(* IEC 61131-3 sources: CS_4_Aufzugsteuerung/src/Stations/CP112/Steuerung/Class/_VaranDriveBase, 1 file *)

(* ---- _VaranDriveBase.st ---- *)
#ifndef _T_VARANDRIVEBASE_H
#define _T_VARANDRIVEBASE_H

#define VAC011_DEVICE_ID		              1005					// device id of VAC011
#define VAC012_DEVICE_ID		              1061					// device id of VAC012
#define VAC013_DEVICE_ID		              1075					// device id of VAC012

#define DIASDRIVE_MAXI_DEVICE_ID          1070          // device id of Dias Drive Maxi
#define DIASDRIVE_MINI_DEVICE_ID          1071          // device id of Dias Drive Mini

//#define DIASDRIVE_WaitTime_ns		            1ms * 1000 * 1000	//time in ns to send next DO in async mode

#define DIASDRIVE_OFFSET_Axis		            16#40							// memory for every axis (offset for axis 1 is 0, for axis 2 is 16#40..)
#define DIASDRIVE_OFFSET_AxisRead	          16#20							//Offset to read data of one axis
#define DIASDRIVE_OFFSET_FAST_AXIS_WRITE    16#C0
#define DIASDRIVE_OFFSET_FAST_AXIS_READ     DIASDRIVE_OFFSET_FAST_AXIS_WRITE + 16#22

#define DIASDRIVE_QUIT_ERROR_WAIT_TIME    50  // in ms

// drive address mapping
#define DIASDRIVE_ADR_ALT_BUF             16#0000  // memory offset for alternating buffer of drive
#define DIASDRIVE_ADR_SERVICE             16#1000  // memory offset for service data of drive
#define DIASDRIVE_ADR_PLL                 16#2000  // memory offset for PLL of drive
#define DIASDRIVE_ADR_LVDS_BUS            16#3000  // memory offset for lvds bus interface of drive
#define DIASDRIVE_ADR_LVDS_DIAG           16#4000  // memory offset for lvds diagnostic of drive

#define DIASDRIVE_ADR_INPUTS              16#4900  // memory offset of digital inputs

#define DIASDRIVE_ADR_OFFSET_CHANNEL      16#0800  // memory for every channel
#define DIASDRIVE_ADR_OFFSET_AXIS         16#0200  // memory for every axis

#define DIASDRIVE_ADR_AXIS_WR_OFFSET      16#0000  // offset to access write data
#define DIASDRIVE_ADR_AXIS_RD_OFFSET      16#0100  // offset to access read data

#define DIASDRIVE_ADR_ALT_BUF_RD_OFFSET   16#0400
#define DIASDRIVE_ADR_ALT_BUF_WR_OFFSET   16#0000

#define DIASDRIVE_ADR_SERVICE_READ        16#0030
#define DIASDRIVE_ADR_SERVICE_WRITE       16#0000

#define DIASDRIVE_MAX_AXIS                8
#define DIASDRIVE_MAX_AXIS_PER_MODULE     3
#define DIASDRIVE_MAX_AXIS_300            3 // with dias drive 300 only up to 3 axis possible

#define WRITETIME_TO_DPRAM                1000 // time in ns to write data to manager dpram

#endif // _T_VARANDRIVEBASE_H

(*!
<Class
	Name               = "_VaranDriveBase"
	Revision           = "1.69"
	RealtimeTask       = "false"
	CyclicTask         = "false"
	BackgroundTask     = "false"
	Sigmatek           = "true"
	OSInterface        = "false"
	HighPriority       = "false"
	Automatic          = "false"
	UpdateMode         = "Prescan"
	IconPath           = ".\Class\Varan_16x16.ico"
	SharedCommandTable = "true"
	Objectsize         = "(584,120)"
	Comment            = "class for VAC011, VAC012 and DiasDrive Mini/Maxi varan interface card">
	<Channels>
		<Server Name="CRC_ErrorCounter" Visualized="true" Initialize="false" WriteProtected="true" Retentive="false" Comment="counts CRC error of all 3 axis"/>
		<Server Name="Input1" Visualized="false" Initialize="false" WriteProtected="true" Retentive="false" Comment="State of digital input 1 of drive&#13;&#10;&#13;&#10;-1..input information not available&#13;&#10; 0..input is low&#13;&#10; 1..input is high"/>
		<Server Name="Input2" Visualized="false" Initialize="false" WriteProtected="true" Retentive="false" Comment="State of digital input 2 of drive&#13;&#10;&#13;&#10;-1..input information not available&#13;&#10; 0..input is low&#13;&#10; 1..input is high"/>
		<Server Name="Input3" Visualized="false" Initialize="false" WriteProtected="true" Retentive="false" Comment="State of digital input 3 of drive&#13;&#10;&#13;&#10;-1..input information not available&#13;&#10; 0..input is low&#13;&#10; 1..input is high"/>
		<Server Name="Input4" Visualized="false" Initialize="false" WriteProtected="true" Retentive="false" Comment="State of digital input 4 of drive&#13;&#10;&#13;&#10;-1..input information not available&#13;&#10; 0..input is low&#13;&#10; 1..input is high"/>
		<Server Name="Input5" Visualized="false" Initialize="false" WriteProtected="true" Retentive="false" Comment="State of digital input 5 of drive&#13;&#10;&#13;&#10;-1..input information not available&#13;&#10; 0..input is low&#13;&#10; 1..input is high"/>
		<Server Name="Input6" Visualized="false" Initialize="false" WriteProtected="true" Retentive="false" Comment="State of digital input 6 of drive&#13;&#10;&#13;&#10;-1..input information not available&#13;&#10; 0..input is low&#13;&#10; 1..input is high"/>
		<Server Name="Input7" Visualized="false" Initialize="false" WriteProtected="true" Retentive="false" Comment="State of digital input 7 of drive&#13;&#10;&#13;&#10;-1..input information not available&#13;&#10; 0..input is low&#13;&#10; 1..input is high"/>
		<Server Name="Input8" Visualized="false" Initialize="false" WriteProtected="true" Retentive="false" Comment="State of digital input 8 of drive&#13;&#10;&#13;&#10;-1..input information not available&#13;&#10; 0..input is low&#13;&#10; 1..input is high"/>
		<Server
			Name           = "RetryCounter"
			Initialize     = "false"
			Visualized     = "true"
			WriteProtected = "true"
			Comment        = "retry counter of varan module">
		</Server>
		<Server
			Name           = "State"
			Initialize     = "false"
			Visualized     = "true"
			WriteProtected = "true">
		</Server>
		<Server Name="Synchron" Visualized="true" Initialize="false" WriteProtected="true" Retentive="false"/>
		<Server Name="VaranOut_1" Class="Hub_Base" Visualized="true" Initialize="false" WriteProtected="true" Retentive="false"/>
		<Client Name="FetchDigitalInputs" Required="false" Internal="false" DefValue="0" Comment="Client is set as init value.&#13;&#10;a value &lt;&gt; 0 means the digital inputs of the drive are fetched synchronously and displayed on the Servers Input1 to Input8"/>
		<Client Name="Hub_Base0" Required="true" Internal="true"/>
		<Client Name="VaranTimeMultiplier" Required="false" Internal="false" Comment="multiplier of varan time as init value."/>
	</Channels>
	<RevDoku>
		<Owner Company="Sigmatek" Author="RamAnd"/>
		<Dokumentation Revision="1.69" Date="16.10.2023" Author="LanSte" Company="Sigmatek" Description="Added GetRequiredWaitTime. If this method is overwritten, the class will wait for for an required module in the init()"/>
		<Dokumentation Revision="1.68" Date="15.06.2022" Author="RamAnd" Company="Sigmatek" Description="Added new Server HardwareVersion to show the hardware version of the VARAN type label."/>
		<Dokumentation Revision="1.67" Date="07.04.2020" Author="EisMic" Company="Sigmatek" Description="Changed comment of client &quot;UserAction&quot; in Varan_Base class."/>
		<Dokumentation Revision="1.66" Date="09.12.2019" Author="LanSte" Company="Sigmatek" Description="Added Server ProtocolVersion. InterframeGap is included in the resource calculation."/>
		<Dokumentation Revision="1.65" Date="30.01.2018" Author="RamAnd" Company="Sigmatek" Description="Class is using constant VM_MULTIVARAN_ADD_DO_INTO_DOL now from VaranManager_Base.h file instead of own define section."/>
		<Dokumentation Revision="1.64" Date="06.02.2017" Author="PieSte" Company="Sigmatek" Description="Changed &quot;Online&quot; server behavior to set online first if cyclic data is valid due to SA35740.&#13;&#10;Corrected an error that MDD100 drives are not initialized if Payload is active."/>
		<Dokumentation Revision="1.63" Date="02.09.2016" Author="ZoePat" Company="Sigmatek" Description="Corrected error with asyncron communication, that could overwrite realtime data for 1 cycle if a SDD3xx was used with VarantimeMultiplier &gt; 1."/>
		<Dokumentation Revision="1.62" Date="10.05.2016" Author="RamAnd" Company="Sigmatek" Description="Suppressed warning that would occur with target ARM on compiler version 30 or higher."/>
		<Dokumentation Revision="1.61" Date="02.05.2016" Author="EisMic" Company="Sigmatek" Description="Corrected an error that SDD115 and SDD120 were not initialized."/>
		<Dokumentation Revision="1.60" Date="04.04.2016" Author="EisMic" Company="Sigmatek" Description="Corrected error in initialisation which leads to an error that the drive is not initialized."/>
		<Dokumentation Revision="1.59" Date="17.02.2016" Author="EisMic" Company="Sigmatek" Description="Prescalersettings were not set correctly when Payload is active."/>
		<Dokumentation Revision="1.58" Date="24.08.2015" Author="EisMic" Company="Sigmatek" Description="DataObjects are now installed in UpdateCy and are added to DOList in UpdateRt if the OS supports the new interface method. Version 16#1003 or higher of the pMultiVaran-Interface is needed to use this feature."/>
		<Dokumentation Revision="1.57" Date="17.06.2015" Author="PieSte" Company="Sigmatek" Description="Corrected function Varan_HwDisconnect() to set dataobjects off."/>
		<Dokumentation Revision="1.56" Date="24.03.2015" Author="EisMic" Company="Sigmatek" Description="Check pointer p_NodeInfo for validity in method GetRetryTimeout due to access exception error if method Varan_HWDisconnect is called and no hardware was available."/>
		<Dokumentation Revision="1.55" Date="30.07.2014" Author="RamAnd" Company="Sigmatek" Description="Loop to check for retries could have caused a crash, if the drive wasn&apos;t initialized so far."/>
		<Dokumentation Revision="1.54" Date="07.07.2014" Author="LanSte" Company="Sigmatek" Description="Added support for reading hardware diagnosis via newinst cmd: CMD_GET_HARDWARE_DIAGNOSE "/>
		<Dokumentation Revision="1.53" Date="04.07.2014" Author="PieSte" Company="Sigmatek" Description="Saved client FetchDigitalInputs to TempFetchDigitalInputs to avoid an access exception if it was changed during run."/>
		<Dokumentation Revision="1.52" Date="07.05.2014" Author="LanSte" Company="Sigmatek" Description="Minimized the interface request via CILGET by useing private pointers to reduce time in init."/>
		<Dokumentation Revision="1.51" Date="06.03.2014" Author="RamAnd" Company="Sigmatek" Description="Changed offset of SyncOut 1 (62,5µs) to be synchron with the SyncOut 0 to prevent inconsistent data in the drive firmware."/>
		<Dokumentation Revision="1.50" Date="12.02.2014" Author="ZoePat" Company="Sigmatek" Description="ExtendedAxis for Axis2 of SDD210 and SDD215 din&apos;t work."/>
		<Dokumentation Revision="1.40" Date="20.01.2014" Author="RamAnd&#13;&#10;PieSte" Company="Sigmatek" Description="Success of GetSyncParameter and SetSyncParameter couldn&apos;t be ensured because the return value wasn&apos;t initialized if the method succeeds.&#13;&#10;Add TaskDelay 15ms in Varan_HwConnect to initialize the Hardware."/>
		<Dokumentation Revision="1.30" Date="05.12.2013" Author="Peeale" Company="Sigmatek" Description="Added payload support; ISO-DOs now start in RT-task to work also on ARM-CPUs;"/>
		<Dokumentation Revision="1.23" Date="18.07.2012" Author="ObeChr" Company="Sigmatek" Description="Implemented time measurement for internal tests in methods UpdateRt, UpdateRtPostScan and UpdateCy"/>
		<Dokumentation Revision="1.22" Date="25.01.2012" Author="ZoePat" Company="Sigmatek" Description="Corrected usage of ENUM types."/>
		<Dokumentation Revision="1.21" Date="09.11.2011" Author="RamAnd" Company="Sigmatek" Description="The memory initialisation of last change has been done too late (after new data was already set)."/>
		<Dokumentation Revision="1.20" Date="16.08.2011" Author="PibPet" Company="Sigmatek" Description="Fixed Problem with the Initialisation from the Drive. Reinit the Memory before sending."/>
		<Dokumentation Revision="1.19" Date="05.07.2011" Author="RamAnd" Company="Sigmatek" Description="Fixed problems in intialisation of SDD drives with less than 3 axis."/>
		<Dokumentation Revision="1.18" Date="14.06.2011" Author="RamAnd" Company="Sigmatek" Description="Fixed crash, when a MDD100 is exchanged with a SDD300 or the other way round."/>
		<Dokumentation Revision="1.17" Date="31.05.2011" Author="RamAnd" Company="Sigmatek" Description="Added possibility to read out the digital inputs of the drive synchronously."/>
		<Dokumentation Revision="1.16" Date="31.05.2011" Author="RamAnd" Company="Sigmatek" Description="DataObjects for VARAN communication are now created and started in the corresponding tasks (ISO-DOs in RT and ASY-DOs in CY) instead of creating and starting all DOs in the connect-callback."/>
		<Dokumentation Revision="1.15" Date="18.05.2011" Author="RamAnd" Company="Sigmatek" Description="After the Online-Server changed to 1, it was possible that the synchron values (like actual position) took 1 more realtime cycle to be shown by the class."/>
		<Dokumentation Revision="1.14" Date="04.01.2011" Author="BleErn" Company="Sigmatek" Description="Added Client Transparent that allows to disable a VARAN-HW-Class"/>
		<Dokumentation Revision="1.13" Date="14.02.2011" Author="BleErn" Company="Sigmatek" Description="Fixed problems with asynchronous communication"/>
		<Dokumentation Revision="1.12" Date="07.12.2010" Author="RamAnd" Company="Sigmatek" Description="Fixed problems in initialisation, when device is plugged in and out within a short time."/>
		<Dokumentation Revision="1.11" Date="25.10.2010" Author="BleErn" Company="Sigmatek" Description="Safety input of VAC013 did not trigger correct errors because of a incorrect comparison of HW-ID"/>
		<Dokumentation Revision="1.10" Date="13.08.2010" Author="BleErn" Company="Sigmatek" Description="Removed an irritating comment from implementation"/>
		<Dokumentation Revision="1.9" Date="10.08.2010" Author="Ramand" Company="Sigmatek" Description="Added support for SDD115"/>
		<Dokumentation Revision="1.8" Date="02.06.2010" Author="BleErn / RamAnd" Company="Sigmatek" Description="Optimization of UpdateRtPostScan method.&#13;&#10;Added support for SDD210"/>
		<Dokumentation Revision="1.7" Date="10.03.2010" Author="RamAnd" Company="Sigmatek" Description="Added serial number validation"/>
		<Dokumentation Revision="1.6" Date="17.05.2010" Author="RamAnd" Company="Sigmatek" Description="Changed defines to avoid compiler warning &quot;Identical Redefinition&quot;"/>
		<Dokumentation Revision="1.5" Date="26.02.2010" Author="RamAnd" Company="Sigmatek" Description="Added support for VAC013"/>
		<Dokumentation Revision="1.4" Date="15.02.2010" Author="RamAnd" Company="Sigmatek" Description="Class works now also with SDD215"/>
		<Dokumentation Revision="1.3" Date="15.01.2010" Author="RamAnd" Company="Sigmatek" Description="Removed Client AxisAvailable. The available axis are now automatically detected."/>
		<Dokumentation Revision="1.2" Date="03.12.2009" Author="RamAnd" Company="Sigmatek" Description="Improved comment on client &quot;AxisAvailable&quot;."/>
		<Dokumentation Revision="1.1" Date="09.11.2009" Author="RamAnd" Company="Sigmatek" Description="Login of VaranRtPostScan did not work properly if the init of the _VaranDriveBase has been called before the VaranManager-Init."/>
		<Dokumentation Revision="1.0" Date="06.10.2009" Author="RamAnd" Company="Sigmatek" Description="Error in Init has been solved (could have led to a VARAN FATAL ERROR)"/>
	</RevDoku>
	<Network Name="_VaranDriveBase">
		<!-- List of Components in this network -->
		<Components>
			<Object
				Name       = "_base"
				Class      = "Varan_Base"
				Position   = "(240,120)"
				Visualized = "true">
				<Channels>
					<Server Name="ConnectCounter"/>
					<Server Name="DeviceAddress"/>
					<Server Name="DeviceID"/>
					<Server Name="DiagControl"/>
					<Server Name="FaultCounter"/>
					<Server Name="HardwareVersion"/>
					<Server Name="Online"/>
					<Server Name="ProtocolVersion"/>
					<Server Name="Release"/>
					<Server Name="RetryCounter"/>
					<Server Name="RXLost"/>
					<Server Name="SerialNo"/>
					<Server Name="State"/>
					<Server Name="TXLost"/>
					<Server Name="ValidateSerNo"/>
					<Server Name="VendorID"/>
					<Client Name="Required" Value="1"/>
					<Client Name="SerNoValidation"/>
					<Client Name="TimeBase" Value="0"/>
					<Client Name="TimeBaseOffset" Value="0"/>
					<Client Name="To_MultiTask"/>
					<Client Name="To_StdLib"/>
					<Client Name="Transparent"/>
					<Client Name="UserAction"/>
					<Client Name="VaranIn"/>
				</Channels>
			</Object>
			<Object
				Name       = "Hub_Base0"
				Class      = "Hub_Base"
				Position   = "(870,780)"
				Visualized = "true">
				<Channels>
					<Server Name="Control"/>
					<Client Name="Splitter_Place" Value="0"/>
					<Client Name="VaranIn"/>
				</Channels>
			</Object>
		</Components>
		<Comments>
		</Comments>
		<!-- List of Connections in this network -->
		<Connections>
			<Connection Source="this.State" Destination="_base.State" Vertices="(1468,210),(724,210),"/>
			<Connection Source="this.Online" Destination="_base.Online" Vertices="(1468,270),(724,270),"/>
			<Connection Source="this.Release" Destination="_base.Release" Vertices="(1468,330),(724,330),"/>
			<Connection Source="this.DeviceAddress" Destination="_base.DeviceAddress" Vertices="(1468,450),(724,450),"/>
			<Connection Source="_base.VaranIn" Destination="this.VaranIn" Vertices="(240,210),(38,210),"/>
			<Connection Source="_base.Required" Destination="this.Required" Vertices="(240,270),(38,270),"/>
			<Connection Source="this.VendorID" Destination="_base.VendorID" Vertices="(1468,510),(724,510),"/>
			<Connection Source="this.DeviceID" Destination="_base.DeviceID" Vertices="(1468,570),(724,570),"/>
			<Connection Source="_base.UserAction" Destination="this.UserAction" Vertices="(240,330),(38,330),"/>
			<Connection Source="Hub_Base0.VaranIn" Destination="_base.State" Vertices="(870,870),(810,870),(810,210),(724,210),"/>
			<Connection Source="this.VaranOut_1" Destination="Hub_Base0.Control" Vertices="(1468,1470),(1296,870),"/>
			<Connection Source="this.RetryCounter" Destination="_base.RetryCounter" Vertices="(1468,690),(724,690),"/>
			<Connection Source="this.Hub_Base0" Destination="Hub_Base0.Control"/>
			<Connection Source="this.SerialNo" Destination="_base.SerialNo" Vertices="(1468,630),(724,630),"/>
			<Connection Source="_base.SerNoValidation" Destination="this.SerNoValidation" Vertices="(240,390),(38,390),"/>
			<Connection Source="this.ValidateSerNo" Destination="_base.ValidateSerNo" Vertices="(1468,750),(724,750),"/>
			<Connection Source="_base.Transparent" Destination="this.Transparent" Vertices="(240,450),(38,450),"/>
			<Connection Source="this.ProtocolVersion" Destination="_base.ProtocolVersion" Vertices="(1468,810),(724,1110),"/>
			<Connection Source="this.HardwareVersion" Destination="_base.HardwareVersion" Vertices="(1468,390),(724,390),"/>
		</Connections>
		<!-- Headerfiles -->
		<Options>
		</Options>
	</Network>
</Class>
*)
#pragma using Varan_Base

_VaranDriveBase : CLASS
: Varan_Base
	TYPE
	  t_AxisState :
	  (
	    _NotUsed,
	    _NoInit,
	    _InitOk,
	    _NoParaList,
	    _NotSynchron,
	    _AxisOk
	  )$USINT;
	  t_ParaState :
	  (
	    _SendExecution,
	    _ResetExecution,
	    _Wait4Response,
	    _IdleState,
	    _GotValueForExecution
	  )$UDINT;
#pragma pack(push, 1)
	  t_ParaList : STRUCT
	    us_number : USINT;
	    sd_value : DINT;
	  END_STRUCT;
#pragma pack(pop)
#pragma pack(push, 1)
	  t_ReadValuePtr : STRUCT  //! <Type Public="true" Name="t_ReadValuePtr"/>
	    a_SyncValues : ARRAY [0..4] OF DINT;
	    bs_InputStates : BSINT
	    [
	      1 OptionBoardInputState,
	    ];
	  END_STRUCT;
#pragma pack(pop)
#pragma pack(push, 1)
	  t_WriteValuePtr : STRUCT  //! <Type Public="true" Name="t_WriteValuePtr"/>
	    a_SyncValues : ARRAY [0..4] OF DINT;
	  END_STRUCT;
#pragma pack(pop)
	  t_AxisData : STRUCT
	    e_AxisState : t_AxisState;
	    us_ParaReady : t_ParaState;
	    sd_Asyncdata : DINT;
	    sd_ObjectError : DINT;
	    b_ListActive : BOOL;
	    p_ParaList : ^t_ParaList;
	    ui_ParaListCnt : UINT;
	    ud_CRCError : UDINT;
	    ud_DOLength : UDINT;
	    b_ExtendedAxis : DINT;
	    b_FastAxis : DINT;
	    b_OldToggleState : DINT;
	    s_ReadValues : t_ReadValuePtr;
	    s_WriteValues : t_WriteValuePtr;
	  END_STRUCT;
#pragma pack(push, 1)
	  t_DataReadOneAxis : STRUCT
	    us_ReceiveState : BSINT
	    [
	      1 ExecutedObjectTransfer,
	      2 CRC_Error,
	      4 OnlineToolWriteOk,
	    ];
	    us_Reserved1 : USINT;
	    us_DigitalIO : USINT;
	    us_TransmitControl : BSINT
	    [
	      1 ToggleBit,
	      2 ErrorInObjectHandling,
	      3 Warning,
	      4 ErrorBit,
	      5 SyncLocked,
	      6 MainsApplied,
	      7 ExternalLock,
	      8 notused,
	    ];
	    sd_ObjectValue : DINT;
	    sd_Value6 : DINT;
	    sd_Value7 : DINT;
	    sd_Value8 : DINT;
	    sd_Value9 : DINT;
	    sd_Value10 : DINT;
	  END_STRUCT;
#pragma pack(pop)
#pragma pack(push, 1)
	  t_DataWriteAsync : STRUCT
	    us_TransmitExecution : BSINT
	    [
	      1 StartObjectTransfer,
	      2 RepeatObjectTransfer,
	      3 EnableValue3_5,
	      4 ClearOnlineToolWriteOk,
	    ];
	    us_Reserved1 : USINT;
	    us_DriveControl : BSINT
	    [
	      1 ToggleBit,
	      2 ReadWriteObject,
	      3 InitCommunicatian,
	      4 EnableInput1,
	      5 UnlockInput1,
	      6 UnlockBrake,
	      7 InterfaceComError,
	      8 NoSetPoint,
	    ];
	    us_ObjectAddress : USINT;
	    sd_ObjectValue : DINT;
	  END_STRUCT;
#pragma pack(pop)
#pragma pack(push, 1)
	  t_DataWriteOneAxis : STRUCT
	    us_TransmitExecution : BSINT
	    [
	      1 StartObjectTransfer,
	      2 RepeatObjectTransfer,
	      3 EnableValue3_5,
	      4 ClearOnlineToolWriteOk,
	    ];
	    us_Reserved1 : USINT;
	    us_DriveControl : BSINT
	    [
	      1 ToggleBit,
	      2 ReadWriteObject,
	      3 InitCommunication,
	      4 EnableInput1,
	      5 UnlockInput1,
	      6 UnlockBrake,
	      7 InterfaceComError,
	      8 NoSetPoint,
	    ];
	    us_ObjectAddress : USINT;
	    sd_ObjectValue : DINT;
	    sd_Value1 : DINT;
	    sd_Value2 : DINT;
	    sd_Value3 : DINT;
	    sd_Value4 : DINT;
	    sd_Value5 : DINT;
	  END_STRUCT;
#pragma pack(pop)
#pragma pack(push, 1)
	  t_FastAxisRead : STRUCT
	    us_DigInOut : USINT;
	    us_TrasmittControl : USINT;
	    sd_Value8 : DINT;
	    sd_Value9 : DINT;
	    sd_Value10 : DINT;
	  END_STRUCT;
#pragma pack(pop)
#pragma pack(push, 1)
	  t_FastAxisWrite : STRUCT
	    us_TransmittExecution : BSINT
	    [
	      5 EnableType2,
	      6 DirectAccess,
	    ];
	    us_Reserved1 : USINT;
	    us_DriveControl : USINT;
	    us_Reserved2 : USINT;
	    sd_Value3 : DINT;
	    sd_Value4 : DINT;
	    sd_Value5 : DINT;
	  END_STRUCT;
#pragma pack(pop)
#pragma pack(push, 1)
	  t_DOFastAxis : STRUCT
	    p_Handle : ^LSL_VARANFRAME;
	    p_DOSettings : ^t_VaranDOSettingsRdWr;
	    p_DataRead : ^t_FastAxisRead;
	    p_DataWrite : ^t_FastAxisWrite;
	    us_OldRetryCounter : USINT;
	  END_STRUCT;
#pragma pack(pop)
	  t_DOOneAxis : STRUCT
	    p_Handle : ^LSL_VARANFRAME;
	    p_DOSettings : ^t_VaranDOSettingsRdWr;
	    p_DataRead : ^t_DataReadOneAxis;
	    p_DataWrite : ^t_DataWriteOneAxis;
	    AsyDataTemp : t_DataWriteOneAxis;
	    b_NewAsyDataTemp : BOOL;
	    us_OldRetryCounter : USINT;
	  END_STRUCT;
#pragma pack(push, 1)
	  t_DrivePLLRd : STRUCT
	    SystemPeriodTime : UINT;
	    Reserved1 : UINT;
	    MaxCountValue : UINT;
	    Reserved2 : UINT;
	    DriveCycleCounter : UINT;
	    StatusRegister : BSINT
	    [
	      1 PLL_Locked,
	    ];
	    Reserved3 : SINT;
	    SyncOut1Offset : UINT;
	    Reserved4 : UINT;
	  END_STRUCT;
#pragma pack(pop)
#pragma pack(push, 1)
	  t_DrivePLLWr : STRUCT
	    SystemPeriodTime : UINT;
	    Reserved1 : UINT;
	  END_STRUCT;
#pragma pack(pop)
	  t_InitSSW :
	  (
	    _SetDataObjectOn,
	    _SetInitAxis,
	    _WaitInit,
	    _SetFinishInit,
	    _SetExecuteBack,
	    _GetFinishInit,
	    _CyIdle
	  )$UDINT;
#pragma pack(push, 1)
	  t_newASYRead : STRUCT
	    sd_ObjectValue : DINT;
	    us_TransmitControl : BSINT
	    [
	      1 ToggleBit,
	      2 ErrorInObjectHandling,
	      3 Warning,
	      4 ErrorBit,
	      5 SyncLocked,
	      6 MainsApplied,
	      7 ExternalLock,
	      8 notused,
	    ];
	    us_DigitalIO : USINT;
	  END_STRUCT;
#pragma pack(pop)
	  t_newASYReadArray : ARRAY [0..DIASDRIVE_MAX_AXIS-1] OF t_newASYRead;
#pragma pack(push, 1)
	  t_newASYWrite : STRUCT
	    sd_ObjectValue : DINT;
	    us_DriveControl : BSINT
	    [
	      1 ToggleBit,
	      2 ReadWriteObject,
	      3 InitCommunication,
	      4 EnableInput1,
	      5 UnlockInput1,
	      6 UnlockBrake,
	      7 InterfaceComError,
	      8 NoSetPoint,
	    ];
	    us_ObjectAddress : USINT;
	  END_STRUCT;
#pragma pack(pop)
	  t_newASYWriteArray : ARRAY [0..DIASDRIVE_MAX_AXIS-1] OF t_newASYWrite;
#pragma pack(push, 1)
	  t_newASYDO : STRUCT
	    p_Handle : ^LSL_VARANFRAME;
	    p_DOSettings : ^t_VaranDOSettingsRdWr;
	    p_DataRead : ^t_newASYReadArray;
	    p_DataWrite : ^t_newASYWriteArray;
	    us_OldRetryCounter : USINT;
	    AsyDataTemp : t_newASYWriteArray;
	    b_NewAsyDataTemp : ARRAY [0..DIASDRIVE_MAX_AXIS-1] OF BOOL;
	  END_STRUCT;
#pragma pack(pop)
#pragma pack(push, 1)
	  t_newDigInDO : STRUCT
	    p_Handle : ^LSL_VARANFRAME;
	    p_DOSettings : ^t_VaranDOSettingsRd;
	    p_DataRead : ^USINT;
	    us_OldRetryCounter : USINT;
	  END_STRUCT;
#pragma pack(pop)
#pragma pack(push, 1)
	  t_newReadDataOneAxis : STRUCT
	    Value6 : DINT;
	    Value7 : DINT;
	    Value8 : DINT;
	    Value9 : DINT;
	    Value10 : DINT;
	  END_STRUCT;
#pragma pack(pop)
#pragma pack(push, 1)
	  t_newWriteDataOneAxis : STRUCT
	    Value1 : DINT;
	    Value2 : DINT;
	    Value3 : DINT;
	    Value4 : DINT;
	    Value5 : DINT;
	  END_STRUCT;
#pragma pack(pop)
#pragma pack(push, 1)
	  t_newISODO : STRUCT
	    p_Handle : ^LSL_VARANFRAME;
	    p_DOSettings : ^t_VaranDOSettingsRdWr;
	    p_DataRead : ^t_newReadDataOneAxis;
	    p_DataWrite : ^t_newWriteDataOneAxis;
	    us_OldRetryCounter : USINT;
	  END_STRUCT;
#pragma pack(pop)
#pragma pack(push, 1)
	  t_ParaSkipOneAxis : STRUCT
	    us_No : USINT;
	    p_Values : ^USINT;
	  END_STRUCT;
#pragma pack(pop)
	  t_ParaSkipList : ARRAY [0..DIASDRIVE_MAX_AXIS-1] OF t_ParaSkipOneAxis;
	  t_RtSSW :
	  (
	    CompInitAxis,
	    CompGetSendParaList,
	    CompWaitForSynchrony,
	    CompOperational,
	    InitAxis,
	    GetSendParaList,
	    WaitForSynchrony,
	    Operational
	  )$UDINT;
	END_TYPE
  //Servers:
	CRC_ErrorCounter 	: SvrCh_DINT;
	Synchron 	: SvrCh_DINT;
	Input1 	: SvrCh_DINT;
	Input2 	: SvrCh_DINT;
	Input3 	: SvrCh_DINT;
	Input4 	: SvrCh_DINT;
	Input5 	: SvrCh_DINT;
	Input6 	: SvrCh_DINT;
	Input7 	: SvrCh_DINT;
	Input8 	: SvrCh_DINT;
	VaranOut_1 	: SvrChCmd_DINT;
  //Clients:
	Hub_Base0 	: CltChCmd_Hub_Base;
	VaranTimeMultiplier 	: CltCh_UDINT;
	FetchDigitalInputs 	: CltCh_DINT;
  //Variables:
		aAxisData : ARRAY [0..DIASDRIVE_MAX_AXIS-1] OF t_AxisData;

		aDataObjects : ARRAY [0..DIASDRIVE_MAX_AXIS-1] OF t_DOOneAxis;

		newIsoDOs : ARRAY [0..DIASDRIVE_MAX_AXIS-1] OF t_newISODO;

		newAsyDO 	: t_newASYDO;
		newDigInDO 	: t_newDigInDO;
		us_Firstscan 	: USINT;
		us_AxisNumber 	: USINT;
		e_InitSSW 	: t_InitSSW;
		b_InitOk 	: BOOL;
		ud_TimemarkInit 	: UDINT;
		ud_TimeCounter 	: UDINT;
		b_SyncEnabled 	: BOOL;
		sd_SyncOffset 	: DINT;
		ud_VaranTime 	: UDINT;
		ud_IsoStartPoint 	: UDINT;
		b_FastDODeactivate 	: BOOL;
		s_DataFastAxis 	: t_DOFastAxis;
		RwFastSpeed 	: t_FastAxisWrite;
		s_SkipParameter 	: t_ParaSkipList;
		AxisAvailableHW : BDINT
		[
		];

		ExtendedAxisSettings : BDINT
		[
		];

		FastAxisSettings : BDINT
		[
		];

		b_CompatibilityMode 	: BOOL;			//! <Variable Comment="TRUE....SDD300 series model&#13;&#10;FALSE...SDD100/5000 series model" Name="b_CompatibilityMode"/>
		pCallBackServer 	: ^UDINT;
		AxisAvailableNo 	: USINT;
		CompAxisAvailableNo 	: SINT;
		AxisAvailable100 	: USINT;
		GetCompAxisSSW 	: UDINT;
		e_RtSSW 	: t_RtSSW;
		CreatedCompDOs 	: BOOL;
		CreatedNewIsoDOs 	: BOOL;
		CreatedNewAsyDOs 	: BOOL;
		b_UpdateThisTime 	: BOOL;
		b_IsSDD21x 	: BOOL;
		b_AlreadyConnected 	: BOOL;
		DataInitFinished 	: BOOL;
		TempFetchDigitalInputs 	: BOOL;
		p_DriveMngBase 	: ^void;
		bAddDOsToListSupport 	: BOOL;			//! <Variable Comment="Flag is True if the os version supports to add DOs to DOL with multivaraninterface (MULTI_VARAN_IINSERTDOINTODOL)" Name="bAddDOsToListSupport"/>
  //Functions:
				//! <Function Comment="=================================================================================================&#13;&#10;Init for Varan Client&#13;&#10;=================================================================================================&#13;&#10;" Name="Init"/>
	FUNCTION VIRTUAL GLOBAL Init;
				//! <Function Comment="Cy - Funktion of Varan class ( called bei VaranMaster )" Name="UpdateCy"/>
	FUNCTION VIRTUAL GLOBAL UpdateCy;
				//! <Function Comment="=================================================================================================&#13;&#10;Rt - Funktion of Varan class ( called bei VaranMaster )&#13;&#10;=================================================================================================&#13;&#10;" Name="UpdateRt"/>
	FUNCTION VIRTUAL GLOBAL UpdateRt;

	FUNCTION VIRTUAL GLOBAL UpdateRtPostScan;
				//! <Function Comment="=================================================================================================&#13;&#10;Function is called if a varan module is connected&#13;&#10;=================================================================================================&#13;&#10;" Name="Varan_HwConnect"/>
	FUNCTION VIRTUAL GLOBAL Varan_HwConnect
		VAR_INPUT
			ud_data 	: UDINT;			//! <Variable Comment="data of call back" Name="Varan_HwConnect.ud_data"/>
		END_VAR
		VAR_OUTPUT
			sd_retval 	: DINT;			//! <Variable Comment="0=Ok, -1=class not okay, -2=wrong axle, -3=axle not in use, -4=varan error in data object" Name="Varan_HwConnect.sd_retval"/>
		END_VAR;
				//! <Function Comment="=================================================================================================&#13;&#10;Function is called if a varan interrupt occures&#13;&#10;=================================================================================================&#13;&#10;" Name="Varan_HwInterrupt"/>
	FUNCTION VIRTUAL GLOBAL Varan_HwInterrupt
		VAR_INPUT
			ud_reason 	: UDINT;			//! <Variable Comment="reason of interrupt" Name="Varan_HwInterrupt.ud_reason"/>
			ud_data 	: ^t_CallBackInterrupt;
		END_VAR
		VAR_OUTPUT
			sd_retval 	: DINT;
		END_VAR;
				//! <Function Comment="=================================================================================================&#13;&#10;Function is called if a varan module is disconnected&#13;&#10;=================================================================================================&#13;&#10;" Name="Varan_HwDisconnect"/>
	FUNCTION VIRTUAL GLOBAL Varan_HwDisconnect
		VAR_INPUT
			ud_data 	: UDINT;
		END_VAR
		VAR_OUTPUT
			sd_retval 	: DINT;
		END_VAR;
				//! <Function Comment="=================================================================================================&#13;&#10;Function to set all Data Objects off&#13;&#10;=================================================================================================&#13;&#10;" Name="SetDOsOff"/>
	FUNCTION VIRTUAL GLOBAL SetDOsOff;
				//! <Function Comment="=================================================================================================&#13;&#10;Function to update module retry counter&#13;&#10;=================================================================================================&#13;&#10;" Name="UpdateRetryCounter"/>
	FUNCTION VIRTUAL GLOBAL UpdateRetryCounter;
				//! <Function Comment="Check if DeviceID is supported by class" Name="CheckDeviceID"/>
	FUNCTION VIRTUAL GLOBAL CheckDeviceID
		VAR_INPUT
			ID2Check 	: UDINT;			//! <Variable Comment="VARAN DeviceID, which should be checked" Name="CheckDeviceID.ID2Check"/>
		END_VAR
		VAR_OUTPUT
			IsOK 	: BOOL;			//! <Variable Comment="TRUE...DeviceID is ok with this class&#13;&#10;FALSE..DeviceID is not ok with this class" Name="CheckDeviceID.IsOK"/>
		END_VAR;
				//! <Function Comment="[#ENGLISH]&#13;&#10;=================================================================================================&#13;&#10;Function to initailize each axle&#13;&#10;=================================================================================================&#13;&#10;[members] s_Axle[x]Data  :R/W :structure for data of one axle&#13;&#10;   s_DataObjectA[x] :R/W :structure for data object of one axle&#13;&#10;   e_InitSSW   :R/W :init ssw&#13;&#10;   ud_TimemarkInit  :W/R :timeout for init&#13;&#10;[locals] p_axle    :W/R :pointer to right axle data&#13;&#10;   p_data_object  :W/R :pointer to right axle data object information&#13;&#10;" Name="InitAxis"/>
	FUNCTION InitAxis
		VAR_INPUT
			us_AxisNo 	: USINT;			//! <Variable Comment="number of axle" Name="InitAxis.us_AxisNo"/>
		END_VAR
		VAR_OUTPUT
			sd_retval 	: DINT;
		END_VAR;
				//! <Function Comment="=================================================================================================&#13;&#10;Function to get object value state&#13;&#10;=================================================================================================&#13;&#10;" Name="GetParameterState"/>
	FUNCTION GLOBAL GetParameterState
		VAR_INPUT
			us_Axis 	: USINT;
		END_VAR
		VAR_OUTPUT
			sd_para_state 	: DINT;			//! <Variable Comment="&gt;0=Object Error, 0=ok, -1=function not ready, -2=wrong axle, -3=Axle not in use, -4=varan error in data object" Name="GetParameterState.sd_para_state"/>
		END_VAR;
				//! <Function Comment="=================================================================================================&#13;&#10;Function to set a object value&#13;&#10;=================================================================================================&#13;&#10;" Name="SetParameter"/>
	FUNCTION GLOBAL SetParameter
		VAR_INPUT
			us_Axis 	: USINT;
			us_para_nr 	: USINT;			//! <Variable Comment="number of parameter" Name="SetParameter.us_para_nr"/>
			us_rdwr 	: USINT;			//! <Variable Comment="0=read, 1=write" Name="SetParameter.us_rdwr"/>
			sd_para_value 	: DINT;			//! <Variable Comment="value of parameter (only for write)" Name="SetParameter.sd_para_value"/>
		END_VAR
		VAR_OUTPUT
			sd_retval 	: DINT;
		END_VAR;
				//! <Function Comment="=================================================================================================&#13;&#10;Function to get object value of parameter&#13;&#10;=================================================================================================&#13;&#10;" Name="GetParameter"/>
	FUNCTION GLOBAL GetParameter
		VAR_INPUT
			us_Axis 	: USINT;
		END_VAR
		VAR_OUTPUT
			sd_para_data 	: DINT;			//! <Variable Comment="value of readed parameter" Name="GetParameter.sd_para_data"/>
		END_VAR;
				//! <Function Comment="=================================================================================================&#13;&#10;Function to set parameter parameter list&#13;&#10;=================================================================================================&#13;&#10;" Name="SetParaList"/>
	FUNCTION GLOBAL SetParaList
		VAR_INPUT
			us_Axis 	: USINT;
			p_list 	: ^void;			//! <Variable Comment="pointer to parameter list" Name="SetParaList.p_list"/>
			ui_counter 	: UINT;			//! <Variable Comment="number of parameters" Name="SetParaList.ui_counter"/>
		END_VAR
		VAR_OUTPUT
			sd_retval 	: DINT;
		END_VAR;
				//! <Function Comment="=================================================================================================&#13;&#10;Function to get a synchron parameter&#13;&#10;=================================================================================================&#13;&#10;" Name="GetSyncParameter"/>
	FUNCTION GLOBAL GetSyncParameter
		VAR_INPUT
			us_Axis 	: USINT;
			us_value 	: USINT;			//! <Variable Comment="0=Value1, 1=Value2, 2=Value3, 3=Value4, 4=Value5" Name="GetSyncParameter.us_value"/>
			p_data 	: ^DINT;			//! <Variable Comment="to this pointer value is written" Name="GetSyncParameter.p_data"/>
		END_VAR
		VAR_OUTPUT
			sd_retval 	: DINT;
		END_VAR;
				//! <Function Comment="=================================================================================================&#13;&#10;Function to set a synchron Parameter&#13;&#10;=================================================================================================&#13;&#10;" Name="SetSyncParameter"/>
	FUNCTION GLOBAL SetSyncParameter
		VAR_INPUT
			us_Axis 	: USINT;
			us_value 	: USINT;
			sd_data 	: DINT;			//! <Variable Comment="data of value" Name="SetSyncParameter.sd_data"/>
		END_VAR
		VAR_OUTPUT
			sd_retval 	: DINT;
		END_VAR;

	FUNCTION InitAxisNew
		VAR_INPUT
			us_AxisNo 	: USINT;
		END_VAR
		VAR_OUTPUT
			sd_retval 	: DINT;
		END_VAR;
				//! <Function Comment="[#ENGLISH]&#13;&#10;=================================================================================================&#13;&#10;Function for parameter handling in synchron mode&#13;&#10;=================================================================================================&#13;&#10;[members] s_Axle[x]Data  :R/W :structure for data of one axle&#13;&#10;   s_DataObjectA[x] :R/W :structure for data object of one axle&#13;&#10;[locals] p_axle   :W/R :pointer to right axle data&#13;&#10;   p_DataObject :W/R :pointer to right data object for axle&#13;&#10;" Name="GetObjectValue"/>
	FUNCTION GetObjectValue
		VAR_INPUT
			us_Axis 	: USINT;
		END_VAR;

	FUNCTION GetObjectValueNew
		VAR_INPUT
			us_Axis 	: USINT;
		END_VAR;
				//! <Function Comment="=================================================================================================&#13;&#10;Function inits drive for all axes used&#13;&#10;=================================================================================================&#13;&#10;" Name="InitDrive"/>
	FUNCTION GLOBAL InitDrive;

	FUNCTION GLOBAL SetAxisOn
		VAR_INPUT
			ud_Axis 	: BDINT;
		END_VAR;
				//! <Function Comment="Function to skip parameters in the parameter list.&#13;&#10;Parameters to be skipped have to be defined via Newinst command 1" Name="SkipEntries"/>
	FUNCTION SkipEntries
		VAR_INPUT
			us_Axis 	: USINT;
			p_Axis 	: ^t_AxisData;
		END_VAR;
				//! <Function Comment="tell the drive class, the software setting and install callback (calls write-method of given server) to get available configuration" Name="StartCommunication"/>
	FUNCTION GLOBAL StartCommunication
		VAR_INPUT
			AxisExtend 	: BDINT;
			AxisFast 	: BDINT;
			pServer4CallBack 	: ^BDINT;			//! <Variable Comment="pass address of server (e.g. #MyServer) to get a callback (write-method) of this server, if the hardware is available on varan (available axis are passed as input parameter)" Name="StartCommunication.pServer4CallBack"/>
		END_VAR;

	FUNCTION GLOBAL GetAxisRdPtr
		VAR_INPUT
			AxisNr 	: DINT;			//! <Variable Comment="number of axis for which you want the pointer (1..8)" Name="GetAxisRdPtr.AxisNr"/>
		END_VAR
		VAR_OUTPUT
			pReadPara 	: ^t_ReadValuePtr;
		END_VAR;

	FUNCTION GLOBAL GetAxisWrPtr
		VAR_INPUT
			AxisNr 	: DINT;
		END_VAR
		VAR_OUTPUT
			pWritePara 	: ^t_WriteValuePtr;
		END_VAR;

	FUNCTION GLOBAL GetDriveIntState
		VAR_OUTPUT
			retcode 	: DINT;			//! <Variable Comment="0..Initialisation of Axles&#13;&#10;1..Download of Drive Parameters&#13;&#10;2..Wait until Drive is synchron with Varan&#13;&#10;3..Operational mode" Name="GetDriveIntState.retcode"/>
		END_VAR;

	FUNCTION GLOBAL ExternInitFinished;

	FUNCTION GetDriveType
		VAR_INPUT
			HWCode 	: DINT;
		END_VAR
		VAR_OUTPUT
			AxisNo 	: SINT;
		END_VAR;

	FUNCTION InstallDefaultDO;

	FUNCTION AddIsoDOsCompMode;

	FUNCTION AddIsoDOsNew;

	FUNCTION GLOBAL GetSeries
		VAR_OUTPUT
			retcode 	: USINT;
		END_VAR;

	FUNCTION GLOBAL IsSDD21x
		VAR_OUTPUT
			retcode 	: BOOL;
		END_VAR;
				//! <Function Comment="Save the passed DriveMngBase this pointer. Needed for Hardwarediagnosis." Name="SetObjectCallBack"/>
	FUNCTION GLOBAL SetObjectCallBack
		VAR_INPUT
			p_DriveMngBaseNew 	: ^void;
		END_VAR;

	FUNCTION VIRTUAL GLOBAL State::NewInst
		VAR_INPUT
			pPara 	: ^CmdStruct;
			pResult 	: ^results;
		END_VAR
		VAR_OUTPUT
			ret_code 	: iprStates;
		END_VAR;
  //Tables:
	FUNCTION @STD
		VAR_OUTPUT
			ret_code	: CONFSTATES;
		END_VAR;
	FUNCTION GLOBAL TAB @CT_;
END_CLASS;

#pragma using Hub_Base

FUNCTION VIRTUAL GLOBAL _VaranDriveBase::Init
  VAR
    sd_retval   : DINT;
  END_VAR

#ifdef IsTransparent_IS_AVAILABLE
  IF IsTransparent() THEN
    return;
  END_IF;
#endif

	//in first init phase
	if ( us_Firstscan = 1 ) then

		//-----------------------------------------------------------------------------------------------
		//init the base class
		Varan_Base::Init();

		//if an error in base class occurs return
		if ( State <> _NotInitialized ) then
			return;
		end_if;

    //Reset Flag
    bAddDOsToListSupport := FALSE;

    //bAddDosToListSupport Flag:
    //Install the isochrone dataobjects in cywork and not in the realtime task, due to the high realtime load in the first rt cycles.
    //The dataobjects are only installed an not added to the DOL in the os with the mask VARAN_DOL_NOT_INSERT_DO_INTO_DOL.
    //With the new os-function MULTI_VARAN_IINSERTDOINTODOL the Dataobjects are now added to the DOL List in the Os.
    //pMultiVaran-Interfaceversion must be equal or higher than 16#1003

    //Check interface version
    if b_PayloadSupport then
      if pMultiVaran then
        if pMultiVaran^.udVersion >= VM_MULTIVARAN_ADD_DO_INTO_DOL then
        // We have the new interface, set flag to remember it later
          bAddDOsToListSupport := TRUE;
        end_if;
      end_if;
    end_if;

    //read cycle time
    VaranTimeMultiplier := VaranTimeMultiplier.read();

    if b_PayloadSupport then
      // Payload DOs automatically use the client Timebase to set the Prescaler of the DOs
      TimeBase := VaranTimeMultiplier;
    end_if;

    if ( VaranTimeMultiplier = 0 ) then
      VaranTimeMultiplier := 1;
    end_if;

    //because on startup we need no waittime for bootloader
    us_AxisNumber := 1;

    //get varan time and calculate offset for sync
    ud_VaranTime := VaranIn.GetVaranTime( #ud_IsoStartPoint );
    sd_SyncOffset := ( ud_VaranTime - ud_IsoStartPoint )$DINT / 10;

    // check if there is a need to get the digital drive inputs
    TempFetchDigitalInputs := (FetchDigitalInputs.Read())$BOOL;
    if TempFetchDigitalInputs = 0 then
      // if not => show that the input information is not available
      Input1 :=
      Input2 :=
      Input3 :=
      Input4 :=
      Input5 :=
      Input6 :=
      Input7 :=
      Input8 := -1;
    end_if;

  elsif us_Firstscan = 2 then // 3rd init, because we need to wait with callback until our pCallBackServer is a valid pointer (done in 2nd init)

    //-----------------------------------------------------------------------------------------------
    //install Varantask
    VaranIn.AddVaranTask( ud_dol_type	:= VARAN_DOL_ISO
              , p_this		:= this
              , callOptions := CALL_OPTION_RT_PRESCAN OR CALL_OPTION_RT_POSTSCAN
              );
    VaranIn.AddVaranTask( ud_dol_type := VARAN_DOL_ASY
                        , p_this      := this
                        );

		//-----------------------------------------------------------------------------------------------
		//call connect hardware function
		sd_retval := Varan_CallBack	( ud_reason	:= VARANMANAGER_CB_CONNECT
                                , ud_data	:= 0
                                );

		//produce Varan Error if module not ok
		if ( sd_retval <> VARANMANAGER_OK ) then

			VaranIn.SetVaranError( p_Node := p_VaranPosition );
		end_if;
  end_if;

	us_Firstscan += 1;

END_FUNCTION

FUNCTION VIRTUAL GLOBAL _VaranDriveBase::Varan_HwConnect
	VAR_INPUT
		ud_data 	: UDINT;
	END_VAR
	VAR_OUTPUT
		sd_retval 	: DINT;
	END_VAR
  VAR
  	i : UDINT;
  END_VAR

	//------------------------------------------------------------------------------------------------
	//get node information
	sd_retval := GetNodeInfo();

	//look for an error
	if ( sd_retval <> VARANMANAGER_OK ) then
		return;
	end_if;

(*
	//look if it is right hardware
	if ((DeviceID <> VAC011_DEVICE_ID )
	&   (DeviceID <> VAC012_DEVICE_ID )
	&   (DeviceID <> VAC013_DEVICE_ID )
  &   (DeviceID <> DIASDRIVE_MINI_DEVICE_ID )
  &   (DeviceID <> DIASDRIVE_MAXI_DEVICE_ID )) then
		State := _WrongHardware;
		return;
  end_if;
*)

  //------------------------------------------------------------------------------------------------
	//we must wait because peripherie reset needs 15ms
	To_MultiTask.TASKDELAY( timeout0 := 15ms );

  // initialize axis data
  for i := 0 to (DIASDRIVE_MAX_AXIS-1) do
    aAxisData[i].e_AxisState := _NotUsed;
  end_for;

  if (DeviceID = VAC011_DEVICE_ID ) |
     (DeviceID = VAC012_DEVICE_ID ) |
     (DeviceID = VAC013_DEVICE_ID ) then
    b_CompatibilityMode := TRUE;
  else
    b_CompatibilityMode := FALSE;
	end_if;

  // reset the write memory of all existing DOs
  // SDD300
  for i := 0 to (sizeof(aDataObjects)/sizeof(t_DOOneAxis))-1 do
    if aDataObjects[i].p_DataWrite then
      _memset(dest:=aDataObjects[i].p_DataWrite, usByte:=0, cntr:=aDataObjects[i].p_DOSettings^.us_ByteCntWr);
    end_if;
  end_for;

  // MDD100
  for i := 0 to (sizeof(newIsoDOs)/sizeof(t_newISODO))-1 do
    if newIsoDOs[i].p_DataWrite then
      _memset(dest:=newIsoDOs[i].p_DataWrite, usByte:=0, cntr:=newIsoDOs[i].p_DOSettings^.us_ByteCntWr);
    end_if;
  end_for;

  // if it's a new drive, check configuration => which axis are available
  if (b_CompatibilityMode = FALSE) then

    //set Pll data (set divider to get 62,5µs)
    //sd_retval :=
    SetNewPllData(ud_delay_time:=0, us_divider:= to_usint(ud_VaranTime / 62500) );
    if b_PayloadSupport then
      sd_retval := MULTI_VARAN_iExecuteDirectAccess(  hNodeHandle := ud_HandleModule
                                                    , udCommand   := VARAN_CMD_MEMORY_READ
                                                    , udOffset    := DIASDRIVE_ADR_SERVICE + 16#60
                                                    , udLength    := sizeof(AxisAvailableHW)
                                                    , pusData     := ( #AxisAvailableHW )$^USINT
                                                    , pudErrorInfo:= NIL);

            //look for an error
      if ( sd_retval <> VARANMANAGER_OK ) then
        State := _DirectAccessFailed;
        return;
      end_if;

    else
      sd_retval := VARAN_iReadMemoryDA(   uiManager		  := ud_VaranManagerNr
                                        , uiAddress		  := DeviceAddress + DIASDRIVE_ADR_SERVICE + 16#60
                                        , uiLen			    := sizeof(AxisAvailableHW)
                                        , uiRetryTimeout:= GetRetryTimeout( ud_bytes := sizeof(AxisAvailableHW) )
                                        , pvData		    := ( #AxisAvailableHW )$^UDINT
                                        , puiError		  := NIL
                                        );

      //look for an error
      if ( sd_retval <> VARANMANAGER_OK ) then
        State := _DirectAccessFailed;
        return;
      end_if;
    end_if;

    // check hw-settings (highest bit is 1 in new version, where hw-configuration is detected)
    if AxisAvailableHW.32 then
      // we delete it, not needed for further use
      AxisAvailableHW.32 := 0;
    else
      AxisAvailableHW := 2#001001011011;  // for older firmware versions, where hw-configuration couldn't be detected
      //           PLACE:  (3)(2)(1)(0)
    end_if;

    e_RtSSW := InitAxis;

    // tell the drive handling class, which of the needed axis are really available
    if pCallBackServer then
      WR(pCallBackServer, AxisAvailableHW$DINT);
    end_if;

  else

    //set Pll data
    sd_retval := SetPllData();

    // in old version there are maximal 3 axis possible, but we don't know how much we got yet
    AxisAvailableHW := 2#111;

    // we don't know how many axis are really available, we have to check parameter with drive info later
    CompAxisAvailableNo := 0;
    GetCompAxisSSW := 0;

    e_RtSSW := CompInitAxis;
  end_if;

  // now we got a connection to the hardware and know which axis are available
  Online := 1;

	//if we are not in init
	if ( us_Firstscan = 12 ) then
		us_AxisNumber := 0;
	end_if;

	//---------------------------------------------------------------------------------------------------------
	//class is not initialized
	ud_TimeCounter 	:= VaranTimeMultiplier;
	b_SyncEnabled 	:= FALSE;
	State			:= _NotInitialized;
	e_InitSSW 		:= _SetDataObjectOn;
	ud_TimemarkInit := ops.tAbsolute;
	sd_retval 		:= VARANMANAGER_OK;

  b_AlreadyConnected := FALSE;

END_FUNCTION

FUNCTION VIRTUAL GLOBAL _VaranDriveBase::Varan_HwInterrupt
	VAR_INPUT
		ud_reason 	: UDINT;
		ud_data 	: ^t_CallBackInterrupt;
	END_VAR
	VAR_OUTPUT
		sd_retval 	: DINT;
	END_VAR
  VAR
  	i : DINT;
  END_VAR

	b_InitOk			:= FALSE;
  b_SyncEnabled := FALSE;
  Online := 0;

	//look if Axis are in use
  for i := 0 to (DIASDRIVE_MAX_AXIS-1) do
    if ( aAxisData[i].e_AxisState <> _NotUsed ) then
      aAxisData[i].e_AxisState := _NoInit;
      aAxisData[i].b_ListActive := FALSE;
      aAxisData[i].us_ParaReady := _IdleState;
    end_if;
  end_for;

  SetDOsOff();

	//call function of base class
	sd_retval := Varan_Base::Varan_HwInterrupt	( ud_reason := ud_reason
                                              , ud_data 	:= ud_data
                                              );

END_FUNCTION

FUNCTION VIRTUAL GLOBAL _VaranDriveBase::Varan_HwDisconnect
	VAR_INPUT
		ud_data 	: UDINT;
	END_VAR
	VAR_OUTPUT
		sd_retval 	: DINT;
	END_VAR
  VAR
  	i : DINT;
  END_VAR

	b_InitOk			:= FALSE;
  b_SyncEnabled := FALSE;
  b_IsSDD21x      := FALSE;
  Online := 0;

	//look if Axis are in use
  for i := 0 to (DIASDRIVE_MAX_AXIS-1) do
    if ( aAxisData[i].e_AxisState <> _NotUsed ) then
      aAxisData[i].e_AxisState := _NoInit;
      aAxisData[i].b_ListActive := FALSE;
      aAxisData[i].us_ParaReady := _IdleState;
    end_if;
  end_for;

  SetDOsOff();

	//call function of base class
	sd_retval := Varan_Base::Varan_HwDisconnect( ud_data := ud_data );

END_FUNCTION

FUNCTION _VaranDriveBase::InitAxis
	VAR_INPUT
		us_AxisNo 	: USINT;
	END_VAR
	VAR_OUTPUT
		sd_retval 	: DINT;
	END_VAR
  VAR
    p_Axis			: ^t_AxisData;
    p_data_object	: ^t_DOOneAxis;
  END_VAR

	//we do this only if class is not initialized
	if ( State <> _NotInitialized ) then
		return;
	end_if;

	//------------------------------------------------------------------------------------------------
	//look which Axis we have and set pointers
//  if (us_AxisNo >= 0) & (us_AxisNo <= (AxisAvailableNo-1)) then
  if (us_AxisNo < DIASDRIVE_MAX_AXIS) & (aAxisData[us_AxisNo].e_AxisState <> _NotUsed) then
    p_Axis			:= #aAxisData[us_AxisNo];
    p_data_object	:= #aDataObjects[us_AxisNo];
  else
    //go to idle state
    sd_retval := _CyIdle;
    return;
  end_if;

	//------------------------------------------------------------------------------------------------
	//look which case we have
	case ( e_InitSSW ) of

		//-----------------------------------------------------------------------------------------------
		_SetDataObjectOn:
					//is Axis in use
					if ( p_Axis^.e_AxisState <> _NotUsed ) then

            if b_PayloadSupport then

              if bAddDOsToListSupport then
                sd_retval := MULTI_VARAN_IINSERTDOINTODOL(p_data_object^.p_Handle$UDINT);
              end_if;

              EnableDO(ud_DOHandle:= p_data_object^.p_Handle$UDINT);
            else
              // Payload DOs automatically use the client Timebase to set the Prescaler of the DOs
            //set right multiplier
              p_data_object^.p_Handle^.ucExePrescaler := VaranTimeMultiplier$USINT - 1;
						//reset data object of Axis
						ResetDataObject	( p_handleDO	:= p_data_object^.p_Handle
                            , us_state		:= VARAN_DO_CONT_RUN
                            , ud_bytes		:= p_Axis^.ud_DOLength * 2
                            );
            end_if;
(*
            if ( us_AxisNo = 3 & UseFastAxis ) then

              ResetDataObject	( p_handleDO	:= s_DataFastAxis.p_Handle
                              , us_state		:= VARAN_DO_CONT_RUN
                              , ud_bytes		:= sizeof( t_FastAxisRead ) + sizeof( t_FastAxisWrite )
                              );

              s_DataFastAxis.p_DataWrite^.us_TransmittExecution.EnableType2 := TRUE;
            end_if;
*)
						//next step
						e_InitSSW := _SetInitAxis;

					else
						//go to idle state
						e_InitSSW := _CyIdle;
					end_if;

		//-----------------------------------------------------------------------------------------------
		_SetInitAxis:
					//InitAxis
					if ( p_Axis^.e_AxisState = _NoInit ) then

						p_data_object^.p_DataWrite^.us_TransmitExecution.StartObjectTransfer 	:= TRUE;
						p_data_object^.p_DataWrite^.us_DriveControl.InitCommunication 			:= TRUE;
					end_if;

					//next step and timestamp
					e_InitSSW 		:= _WaitInit;
					ud_TimemarkInit := ops.tAbsolute;

		//-----------------------------------------------------------------------------------------------
		_WaitInit:	//reset startobjecttransfer bit
					p_data_object^.p_DataWrite^.us_TransmitExecution.StartObjectTransfer 	:= FALSE;

					//look if Axis 1 must be init
					if ( p_Axis^.e_AxisState = _NoInit ) then

						//object must be executed, error in object handling must be set and error code must be 9
						if	( p_data_object^.p_DataRead^.us_ReceiveState.ExecutedObjectTransfer		= TRUE
							& p_data_object^.p_DataRead^.us_TransmitControl.ErrorInObjectHandling	= TRUE
							& p_data_object^.p_DataRead^.sd_ObjectValue 							= 9
							)
						then
							//set Axis to next state
							p_Axis^.e_AxisState := _NoParaList;
							e_InitSSW := _SetFinishInit;
            //after timeout check again
            elsif ( ops.tAbsolute - ud_TimemarkInit > 1sec ) then
              e_InitSSW := _SetInitAxis;
            end_if;
          //after timeout check again
					elsif ( ops.tAbsolute - ud_TimemarkInit > 1sec ) then
						e_InitSSW := _SetInitAxis;
					end_if;

		//-----------------------------------------------------------------------------------------------
		_SetFinishInit:

					//If Axis is in right state
					if ( p_Axis^.e_AxisState = _NoParaList ) then

						p_data_object^.p_DataWrite^.us_TransmitExecution.StartObjectTransfer 	:= TRUE;
						p_data_object^.p_DataWrite^.us_DriveControl.InitCommunication 			:= FALSE;
					end_if;

					//next step and timestamp
					e_InitSSW 		:= _GetFinishInit;
					ud_TimemarkInit := ops.tAbsolute;

		//-----------------------------------------------------------------------------------------------
		_GetFinishInit:

					//look if Axis is in use and error bit is reset
					if	( p_data_object^.p_DataRead^.us_TransmitControl.ErrorInObjectHandling = FALSE) &
						  ( p_data_object^.p_DataRead^.us_ReceiveState.ExecutedObjectTransfer 	= TRUE )
					then
					//reset startobjecttransfer bit
            p_data_object^.p_DataWrite^.us_TransmitExecution.StartObjectTransfer 	:= FALSE;

						//final step, init ok and class ok
						e_InitSSW := _CyIdle;

					else

						//try again if return value is 10 or 8 (see DiasDrive Doku)
						if	( ( p_data_object^.p_DataRead^.sd_ObjectValue = 10 | p_data_object^.p_DataRead^.sd_ObjectValue = 8 )
							& p_data_object^.p_DataRead^.us_TransmitControl.ErrorInObjectHandling = TRUE
							)
						then
							e_InitSSW 			:= _SetInitAxis;
							p_Axis^.e_AxisState := _NoInit;
						end_if;

						//if timeout check again
						if ( ops.tAbsolute - ud_TimemarkInit > 2sec ) then
							e_InitSSW := _SetFinishInit;
						end_if;
					end_if;

		//-----------------------------------------------------------------------------------------------
		_CyIdle:

	end_case;

	//return ssw
	sd_retval := e_InitSSW$DINT;

END_FUNCTION

FUNCTION VIRTUAL GLOBAL _VaranDriveBase::UpdateRt
  VAR
    sd_retval		: DINT;
    i           : UDINT;
    TempInputs  : BSINT;
  END_VAR

//=================================================================================================
#ifdef VM_CLASS_TIME_MEASUREMENT
	StartTimeMeasurement(VARANTIME_RT);
#endif
//=================================================================================================

	//update in right intervall
	ud_TimeCounter -= 1;
	if ( ud_TimeCounter <> 0 ) THEN
    b_UpdateThisTime := FALSE;
		return;
  else
    b_UpdateThisTime := TRUE;
	end_if;

	ud_TimeCounter := VaranTimeMultiplier;

	//call rt of base
	Varan_Base::UpdateRt();

  if Online then
    case e_RtSSW of

      //*****************************************************************************
      //**      Comp = compatibility mode to dias drive 300 series                 **
      //*****************************************************************************
      CompInitAxis:

        //first enable sync of varan and drive
        if ( b_SyncEnabled = FALSE ) then
          sd_retval := EnableSyncOut	( us_sync_nr				:= 0
                                      , sd_offset					:= sd_SyncOffset
                                      , us_period_multiplier		:= VaranTimeMultiplier$USINT
                                      , us_frame_count_treshold	:= 0
                                      , us_enable_frame_count		:= 0
                                      , b_use_divider_sync := FALSE
                                      );

          //look for an error
          if ( sd_retval <> VARANMANAGER_OK ) then
            return;
          end_if;

          sd_retval := EnableSyncOut	( us_sync_nr				:= 1
                                      , sd_offset					:= sd_SyncOffset MOD 6250
                                      , us_period_multiplier		:= 0
                                      , us_frame_count_treshold	:= 0
                                      , us_enable_frame_count		:= 0
                                      , b_use_divider_sync := TRUE
                                      );

          //look for an error
          if ( sd_retval <> VARANMANAGER_OK ) then
            return;
          end_if;

          b_SyncEnabled := TRUE;
          return;
        end_if;

        if bAddDOsToListSupport = false then
          InstallDefaultDO();
        end_if;

        if b_AlreadyConnected = TRUE then
          //*****************************************************************************
          //**  switch Axis                                                            **
          //*****************************************************************************
          case ( us_AxisNumber ) of

            // ***********************************************************************************************************************************
            0:	//we must wait 3 secs because in sdrive bootloader is active
                  if ( ops.tAbsolute - ud_TimemarkInit > 3secs ) then
                    us_AxisNumber += 1;
                  end_if;

            // ***********************************************************************************************************************************
            1: 	//wait until first axis is initialized
                if InitAxis( us_AxisNo := 0 ) = _CyIdle$DINT then
                  us_AxisNumber 	+=1;
                  e_InitSSW 	:= _SetDataObjectOn;
                end_if;

            // ***********************************************************************************************************************************
            2: // we check how many axis are really available (parameter communication)
              //Check for DataInitFinished false too, because CompAxisAvailableNo is changed in step 1 so step 2 of the ssw would not be executed
              if CompAxisAvailableNo = 0 | DataInitFinished = FALSE  then
                case GetCompAxisSSW of

                  // ***********************************************************************************************************************************
                  0:
                    //set data for object handling
                    aAxisData[0].us_ParaReady := _SendExecution;

                    aDataObjects[0].p_DataWrite^.us_ObjectAddress	:= 189;
                    aDataObjects[0].p_DataWrite^.sd_ObjectValue		:= 0;
                    aDataObjects[0].p_DataWrite^.us_DriveControl.ReadWriteObject := 0;

                    GetCompAxisSSW += 1;

                  // ***********************************************************************************************************************************
                  1:
                    //Axis "0" object value
                    GetObjectValue( us_Axis := 0 );

                    //look if parameter handling is ready
                    if	( aAxisData[0].us_ParaReady	= _IdleState ) &
                        ( aAxisData[0].b_ListActive	= FALSE)  &
                        ( aDataObjects[0].p_DataWrite^.us_ObjectAddress = 189) then
                      //look for an object handling error
                      if (aAxisData[0].sd_ObjectError = 0) then
                        sd_retval := GetParameter(us_axis:=0);
                        if sd_retval <> 120 then
                          CompAxisAvailableNo := GetDriveType(sd_retval);
                          if CompAxisAvailableNo > 0 then
                            AxisAvailableNo := CompAxisAvailableNo$USINT;
                          end_if;

                          // at SDD215 the middle axis is not available
                          if b_IsSDD21x then
                            aAxisData[1].e_AxisState := _NotUsed;
                          end_if;

                          // tell the drive handling class, which of the needed axis are really available
                          if pCallBackServer then
                            WR(pCallBackServer, AxisAvailableHW$DINT);
                          end_if;

                          DataInitFinished := FALSE;
                          GetCompAxisSSW += 1;

                        else
                          GetCompAxisSSW := 0;
                        end_if;
                      end_if;
                    end_if;

                  // ***********************************************************************************************************************************
                  2:	//is done at cy task if bAddDOsToListSupport is true

                    //Check if we can use the new interface and add DOs in UpdateCy
                    if bAddDOsToListSupport = false then
                      //We have the old interface, install DOs here
                      AddIsoDOsCompMode();
                    end_if;

                end_case;

              else

                if us_AxisNumber <= AxisAvailableNo then
                  if AxisAvailableHW AND (1 SHL (us_AxisNumber-1)$UDINT) then
                    if InitAxis( us_AxisNo := us_AxisNumber-1 ) = _CyIdle$DINT then
                      us_AxisNumber += 1;
                      e_InitSSW 	:= _SetDataObjectOn;
                    end_if;
                  else
                    us_AxisNumber += 1;
                  end_if;
                else
                  us_AxisNumber := DIASDRIVE_MAX_AXIS_300+1;
                end_if;
              end_if;

            // ***********************************************************************************************************************************
            3..DIASDRIVE_MAX_AXIS_300:
              if us_AxisNumber <= AxisAvailableNo then
                if AxisAvailableHW AND (1 SHL (us_AxisNumber-1)$UDINT) then
                  if InitAxis( us_AxisNo := us_AxisNumber-1 ) = _CyIdle$DINT then
                    us_AxisNumber += 1;
                    e_InitSSW 	:= _SetDataObjectOn;
                  end_if;
                else
                  us_AxisNumber += 1;
                end_if;
              else
                us_AxisNumber := DIASDRIVE_MAX_AXIS_300+1;
              end_if;

            else
              //class is ready
              b_InitOk 	:= TRUE;
              us_AxisNumber 	:= 0;
              e_RtSSW := CompGetSendParaList;

          end_case;

        end_if;

      // ******************************************************************************************************************************************
      CompGetSendParaList:

        // update asynchron parameters
        sd_retval := 0;
        if AxisAvailableNo then
          for i := 0 to (AxisAvailableNo-1) do
            // at SDD215 the middle axis is not available
            if aAxisData[i].e_AxisState <> _NotUsed then
              //Axis "i" object value
              GetObjectValue( us_Axis := to_usint(i) );
            end_if;
          end_for;
        end_if;

      // we get into the next step via ExternInitFinished-Method
      // ******************************************************************************************************************************************

      CompWaitForSynchrony:
        if AxisAvailableNo & aDataObjects[0].p_DataRead^.us_TransmitControl.SyncLocked then
          // before we set state to operational we get the values 1 time otherwise online would be 1 but no actual values are available
          for i := 0 to (AxisAvailableNo-1) do
            if ( aAxisData[i].e_AxisState <> _NotUsed ) then
              aAxisData[i].e_AxisState := _AxisOk;

              //-----------------------------------------------------------------------------------------------
              // update asynchron parameters
              //Axis "i" object value
              GetObjectValue( us_Axis := to_usint(i) );
              //------------------------------------------------------------------------------------------------

              if aAxisData[i].b_ExtendedAxis then
                _memcpy(#aAxisData[i].s_ReadValues.a_SyncValues[ 0 ], #aDataObjects[i].p_DataRead^.sd_Value6, 5 * sizeof(DINT));
              else
                aAxisData[i].s_ReadValues.a_SyncValues[ 0 ] := aDataObjects[i].p_DataRead^.sd_Value6;
                aAxisData[i].s_ReadValues.a_SyncValues[ 1 ] := aDataObjects[i].p_DataRead^.sd_Value7;

              end_if;

              //look for CRC error
              if ( aDataObjects[i].p_DataRead^.us_ReceiveState.CRC_Error = TRUE ) then
                aAxisData[i].ud_CRCError += 1;
                CRC_ErrorCounter += 1;
              end_if;
            end_if;
          end_for;

          e_RtSSW := CompOperational;
          State 		:= _ClassOk;
        end_if;

      // ******************************************************************************************************************************************
      CompOperational:
        if AxisAvailableNo then
          Synchron := aDataObjects[0].p_DataRead^.us_TransmitControl.SyncLocked;
          if Synchron then
            for i := 0 to (AxisAvailableNo-1) do
              if ( aAxisData[i].e_AxisState <> _NotUsed ) then
                aAxisData[i].e_AxisState := _AxisOk;

                //-----------------------------------------------------------------------------------------------
                // update asynchron parameters
                //Axis "i" object value
                GetObjectValue( us_Axis := to_usint(i) );
                //------------------------------------------------------------------------------------------------

                if aAxisData[i].b_ExtendedAxis then
                  _memcpy(#aAxisData[i].s_ReadValues.a_SyncValues[ 0 ], #aDataObjects[i].p_DataRead^.sd_Value6, 5 * sizeof(DINT));
                else
                  aAxisData[i].s_ReadValues.a_SyncValues[ 0 ] := aDataObjects[i].p_DataRead^.sd_Value6;
                  aAxisData[i].s_ReadValues.a_SyncValues[ 1 ] := aDataObjects[i].p_DataRead^.sd_Value7;

                end_if;

                //look for CRC error
                if ( aDataObjects[i].p_DataRead^.us_ReceiveState.CRC_Error = TRUE ) then
                  aAxisData[i].ud_CRCError += 1;
                  CRC_ErrorCounter += 1;
                end_if;
              end_if;
            end_for;
          else
            for i := 0 to (AxisAvailableNo-1) do
              if ( aAxisData[i].e_AxisState <> _NotUsed ) then
                aAxisData[i].e_AxisState := _NotSynchron;

                //-----------------------------------------------------------------------------------------------
                // update asynchron parameters
                //Axis "i" object value
                GetObjectValue( us_Axis := to_usint(i) );
                //------------------------------------------------------------------------------------------------

                if aAxisData[i].b_ExtendedAxis then
                  _memcpy(#aAxisData[i].s_ReadValues.a_SyncValues[ 0 ], #aDataObjects[i].p_DataRead^.sd_Value6, 5 * sizeof(DINT));
                else
                  aAxisData[i].s_ReadValues.a_SyncValues[ 0 ] := aDataObjects[i].p_DataRead^.sd_Value6;
                  aAxisData[i].s_ReadValues.a_SyncValues[ 1 ] := aDataObjects[i].p_DataRead^.sd_Value7;
                end_if;

                //look for CRC error
                if ( aDataObjects[i].p_DataRead^.us_ReceiveState.CRC_Error = TRUE ) then
                  aAxisData[i].ud_CRCError += 1;
                  CRC_ErrorCounter += 1;
                end_if;
              end_if;
            end_for;
          end_if;
        end_if;

      // ******************************************************************************************************************************************
      // now the part for DiasDrive 100/5000 series
      // ******************************************************************************************************************************************
      // ******************************************************************************************************************************************
      InitAxis:

        if bAddDOsToListSupport = false then
          AddIsoDOsNew();
        end_if;

        //Check if Hardware is already connected (DOs created)
        if b_AlreadyConnected & e_InitSSW = _SetDataObjectOn then

        //switch Axis
          case ( us_AxisNumber ) of

            0:	//we must wait 3 secs because in sdrive bootloader is active
              if ( ops.tAbsolute - ud_TimemarkInit > 3secs ) then
                us_AxisNumber += 1;
              end_if;

            1..DIASDRIVE_MAX_AXIS: 	//wait until Axis are initialized
              if us_AxisNumber <= AxisAvailableNo then
                if InitAxisNew( us_AxisNo := us_AxisNumber-1 ) = _CyIdle$DINT then
                  us_AxisNumber 	+=1;
                  e_InitSSW 	:= _SetDataObjectOn;
                end_if;
              else
                us_AxisNumber := DIASDRIVE_MAX_AXIS+1;
              end_if;

            else
              //class is ready
              b_InitOk 	:= TRUE;
              us_AxisNumber 	:= 0;
              e_RtSSW := GetSendParaList;

          end_case;
        end_if;

      // ******************************************************************************************************************************************
      WaitForSynchrony:
      //#pragma message("Synchronität wird bei DiasDrive 100/5000 testweise noch nicht überprüft!")
      // evtl. asynchrones DO deaktivieren, wenn keine asynchronen Daten übertragen werden,
      // kann aber erst mit finalem Mapping entschieden werden, da vielleicht noch IOs dazukommen

  //      if AxisAvailableNo & newAsyDO.p_DataRead^[0].us_TransmitControl.SyncLocked then

          // before we set state to operational we get the values 1 time otherwise online would be 1 but no actual values are available
          if AxisAvailableNo then
            Synchron := 1;//newAsyDO.p_DataRead^[0].us_TransmitControl.SyncLocked;
            if Synchron then
              for i := 0 to (AxisAvailableNo-1) do
                if ( aAxisData[i].e_AxisState <> _NotUsed ) then
                  aAxisData[i].e_AxisState := _AxisOk;

                  if aAxisData[i].b_ExtendedAxis then
                    _memcpy(#aAxisData[i].s_ReadValues.a_SyncValues[ 0 ], #newIsoDOs[i].p_DataRead^.Value6, sizeof(t_newReadDataOneAxis));
                  else
                    aAxisData[i].s_ReadValues.a_SyncValues[ 0 ] := newIsoDOs[i].p_DataRead^.Value6;
                    aAxisData[i].s_ReadValues.a_SyncValues[ 1 ] := newIsoDOs[i].p_DataRead^.Value7;
                  end_if;
                end_if;
              end_for;
            else
              for i := 0 to (AxisAvailableNo-1) do
                if ( aAxisData[i].e_AxisState <> _NotUsed ) then
                  aAxisData[i].e_AxisState := _NotSynchron;

                  if aAxisData[i].b_ExtendedAxis then
                    _memcpy(#aAxisData[i].s_ReadValues.a_SyncValues[ 0 ], #newIsoDOs[i].p_DataRead^.Value6, sizeof(t_newReadDataOneAxis));
                  else
                    aAxisData[i].s_ReadValues.a_SyncValues[ 0 ] := newIsoDOs[i].p_DataRead^.Value6;
                    aAxisData[i].s_ReadValues.a_SyncValues[ 1 ] := newIsoDOs[i].p_DataRead^.Value7;
                  end_if;
                end_if;
              end_for;
            end_if;
          end_if;

          if TempFetchDigitalInputs then
            TempInputs := newDigInDO.p_DataRead^;
            Input1 := TempInputs.1;
            Input2 := TempInputs.2;
            Input3 := TempInputs.3;
            Input4 := TempInputs.4;
            Input5 := TempInputs.5;
            Input6 := TempInputs.6;
            Input7 := TempInputs.7;
            Input8 := TempInputs.8;
          end_if;

          e_RtSSW := Operational;
          State 		:= _ClassOk;
  //      end_if;

      // ******************************************************************************************************************************************
      Operational:

        if AxisAvailableNo then
          Synchron := 1;//newAsyDO.p_DataRead^[0].us_TransmitControl.SyncLocked;
          if Synchron then
            for i := 0 to (AxisAvailableNo-1) do
              if ( aAxisData[i].e_AxisState <> _NotUsed ) then
                aAxisData[i].e_AxisState := _AxisOk;

                if aAxisData[i].b_ExtendedAxis then
                  _memcpy(#aAxisData[i].s_ReadValues.a_SyncValues[ 0 ], #newIsoDOs[i].p_DataRead^.Value6, sizeof(t_newReadDataOneAxis));
                else
                  aAxisData[i].s_ReadValues.a_SyncValues[ 0 ] := newIsoDOs[i].p_DataRead^.Value6;
                  aAxisData[i].s_ReadValues.a_SyncValues[ 1 ] := newIsoDOs[i].p_DataRead^.Value7;
                end_if;
              end_if;
            end_for;
          else
            for i := 0 to (AxisAvailableNo-1) do
              if ( aAxisData[i].e_AxisState <> _NotUsed ) then
                aAxisData[i].e_AxisState := _NotSynchron;

                if aAxisData[i].b_ExtendedAxis then
                  _memcpy(#aAxisData[i].s_ReadValues.a_SyncValues[ 0 ], #newIsoDOs[i].p_DataRead^.Value6, sizeof(t_newReadDataOneAxis));
                else
                  aAxisData[i].s_ReadValues.a_SyncValues[ 0 ] := newIsoDOs[i].p_DataRead^.Value6;
                  aAxisData[i].s_ReadValues.a_SyncValues[ 1 ] := newIsoDOs[i].p_DataRead^.Value7;
                end_if;
              end_if;
            end_for;
          end_if;
        end_if;

        if TempFetchDigitalInputs then
          TempInputs := newDigInDO.p_DataRead^;
          Input1 := TempInputs.1;
          Input2 := TempInputs.2;
          Input3 := TempInputs.3;
          Input4 := TempInputs.4;
          Input5 := TempInputs.5;
          Input6 := TempInputs.6;
          Input7 := TempInputs.7;
          Input8 := TempInputs.8;
        end_if;

    end_case;
  end_if;
(*
    if ( UseFastAxis ) then
      s_DataFastAxis.p_DataWrite^.sd_Value3 := Axis3_Speed;

      //activate DO if deactivated
      if ( b_FastDODeactivate ) then
        b_FastDODeactivate := FALSE;
        s_DataFastAxis.p_DataWrite^.us_TransmittExecution.DirectAccess := FALSE;

        ResetDataObject ( p_handleDO  := s_DataFastAxis.p_Handle
                        , us_state    := VARAN_DO_CONT_RUN
                        , ud_bytes    := sizeof( t_FastAxisRead ) + sizeof( t_FastAxisWrite )
                        );
      end_if;

    else
*)

//=================================================================================================
#ifdef VM_CLASS_TIME_MEASUREMENT
	StopTimeMeasurement(VARANTIME_RT);
#endif
//=================================================================================================
END_FUNCTION

FUNCTION _VaranDriveBase::GetObjectValue
	VAR_INPUT
		us_Axis 	: USINT;
	END_VAR
  VAR
    p_Axis			: ^t_AxisData;
    p_DataObject	: ^t_DOOneAxis;
  END_VAR

	//------------------------------------------------------------------------------------------------
	//look which Axis we have and set pointers
//  if (us_Axis >= 0) & (us_Axis <= (AxisAvailableNo-1)) then
  if (us_Axis < DIASDRIVE_MAX_AXIS) & (aAxisData[us_Axis].e_AxisState <> _NotUsed) then
    p_Axis			:= #aAxisData[us_Axis];
    p_DataObject	:= #aDataObjects[us_Axis];
  else
    //else do nothing (should not come here)
    return;
  end_if;

	//------------------------------------------------------------------------------------------------
	//get to right step
	case ( p_Axis^.us_ParaReady ) of

		_SendExecution:		//send transmit execution request for object handling
							p_DataObject^.p_DataWrite^.us_TransmitExecution.StartObjectTransfer := TRUE;

//              p_Axis^.b_OldToggleState := p_DataObject^.p_DataRead^.us_TransmitControl.ToggleBit;

              p_DataObject^.p_DataWrite^.us_DriveControl.ToggleBit := NOT p_DataObject^.p_DataWrite^.us_DriveControl.ToggleBit;

							//reset error and go to next step
							p_Axis^.sd_ObjectError := 0;
							p_Axis^.us_ParaReady := _ResetExecution;

		_ResetExecution:	//reset transmit execution request bit

              if (p_DataObject^.p_DataRead^.us_ReceiveState.ExecutedObjectTransfer = FALSE) then
                p_DataObject^.p_DataWrite^.us_TransmitExecution.StartObjectTransfer := FALSE;
                p_Axis^.us_ParaReady := _Wait4Response;
              end_if;

		_Wait4Response:		//wait until receive state is true
							if ( p_DataObject^.p_DataRead^.us_ReceiveState.ExecutedObjectTransfer = TRUE ) then// &
                 //( p_DataObject^.p_DataRead^.us_TransmitControl.ToggleBit <> p_Axis^.b_OldToggleState) then

								//look if we have a parameter list
								if ( p_Axis^.b_ListActive = TRUE ) then

                  // skip all defined parameter entries
                  SkipEntries(us_Axis, p_Axis);

									//have we set all parameter
									if ( p_Axis^.ui_ParaListCnt ) then

										//set data to object handling registers
										p_DataObject^.p_DataWrite^.us_ObjectAddress					:= p_Axis^.p_ParaList^.us_number;
										p_DataObject^.p_DataWrite^.sd_ObjectValue					:= p_Axis^.p_ParaList^.sd_value;
										p_DataObject^.p_DataWrite^.us_DriveControl.ReadWriteObject	:= TRUE;

										//set next parameter step and set pointer to next parameter data
										p_Axis^.us_ParaReady 	:= _SendExecution;
										p_Axis^.ui_ParaListCnt 	-= 1;
										p_Axis^.p_ParaList 		+= sizeof( t_ParaList );

									else
										//set ssw to idle and deactivate parameter list
										p_Axis^.b_ListActive 	:= FALSE;

										//look if we get a parameter list
										if ( p_Axis^.e_AxisState = _NoParaList ) then
											p_Axis^.e_AxisState		:= _NotSynchron;
										end_if;

										p_Axis^.us_ParaReady 	:= _IdleState;

									end_if;

								else
									//get to idle step
									p_Axis^.us_ParaReady := _IdleState;

									//look for an object error
									if ( p_DataObject^.p_DataRead^.us_TransmitControl.ErrorInObjectHandling = TRUE ) then
										p_Axis^.sd_ObjectError := p_DataObject^.p_DataRead^.sd_ObjectValue;
									else
                 		p_Axis^.sd_Asyncdata := p_DataObject^.p_DataRead^.sd_ObjectValue;
                  end_if;

								end_if;
							end_if;

		_IdleState:				//do nothing in this step

	end_case;

END_FUNCTION

FUNCTION GLOBAL _VaranDriveBase::SetParameter
	VAR_INPUT
		us_Axis 	: USINT;
		us_para_nr 	: USINT;
		us_rdwr 	: USINT;
		sd_para_value 	: DINT;
	END_VAR
	VAR_OUTPUT
		sd_retval 	: DINT;
	END_VAR
  VAR
    p_Axis			: ^t_AxisData;
    p_data_object	: ^t_DOOneAxis;
    p_Write     : ^t_newASYWrite;
  END_VAR

	sd_retval := -1;

	//look if class is ok
	if ( State <> _ClassOk ) & ( GetDriveIntState()$t_RtSSW <> CompGetSendParaList ) then
		return;
	end_if;

	//look if init was ok
	if ( b_InitOk ) then

    // if it's a SDD300 model
    if b_CompatibilityMode then

      //------------------------------------------------------------------------------------------------
      //look which Axis we have and set pointers
//      if (us_Axis >= 0) & (us_Axis <= (AxisAvailableNo-1)) then
      if (us_Axis < DIASDRIVE_MAX_AXIS) & (aAxisData[us_Axis].e_AxisState <> _NotUsed) then
        p_Axis			:= #aAxisData[us_Axis];
        p_data_object	:= #aDataObjects[us_Axis];
      else
        sd_retval := -2;
        return;
      end_if;

      //----------------------------------------------------------------------------------------------
      //look if Axis is in use
      if ( p_Axis^.e_AxisState = _NotUsed ) then
        sd_retval := -3;
        return;
      end_if;

      //look if parameter handling is ready
      if	( p_Axis^.us_ParaReady = _IdleState
        & p_Axis^.b_ListActive = FALSE
        )
      then

        //set data for object handling
        p_Axis^.us_ParaReady := _GotValueForExecution;
//        p_data_object^.AsyDataTemp := aDataObjects[us_Axis].p_DataWrite^;
        p_data_object^.AsyDataTemp.us_ObjectAddress	:= us_para_nr;
        p_data_object^.AsyDataTemp.sd_ObjectValue		:= sd_para_value;

        if ( us_RdWr ) then
          p_data_object^.AsyDataTemp.us_DriveControl.ReadWriteObject := 1;
        else
          p_data_object^.AsyDataTemp.us_DriveControl.ReadWriteObject := 0;
        end_if;

        p_data_object^.b_NewAsyDataTemp := TRUE;

        sd_retval := 0;
      end_if;
    else
    // if it's a SDD100/5000 model

      //------------------------------------------------------------------------------------------------
      //look which Axis we have and set pointers
//      if (us_Axis >= 0) & (us_Axis <= (AxisAvailableNo-1)) then
      if (us_Axis < DIASDRIVE_MAX_AXIS) & (aAxisData[us_Axis].e_AxisState <> _NotUsed) then
        p_Axis			:= #aAxisData[us_Axis];
        p_Write := #newAsyDO.AsyDataTemp[us_Axis];
      else
        sd_retval := -2;
        return;
      end_if;

      //----------------------------------------------------------------------------------------------
      //look if Axis is in use
      if ( p_Axis^.e_AxisState = _NotUsed ) then
        sd_retval := -3;
        return;
      end_if;

      //look if parameter handling is ready
      if	( p_Axis^.us_ParaReady = _IdleState
        & p_Axis^.b_ListActive = FALSE
        )
      then

        //set data for object handling
        p_Axis^.us_ParaReady := _GotValueForExecution;
        p_Write^ := newAsyDO.p_DataWrite^[us_Axis];
        p_Write^.us_ObjectAddress	:= us_para_nr;
        p_Write^.sd_ObjectValue		:= sd_para_value;

        if ( us_RdWr ) then
          p_Write^.us_DriveControl.ReadWriteObject := 1;
        else
          p_Write^.us_DriveControl.ReadWriteObject := 0;
        end_if;

        newAsyDO.b_NewAsyDataTemp[us_Axis] := TRUE;

        sd_retval := 0;
      end_if;
    end_if;
	end_if;

END_FUNCTION

FUNCTION GLOBAL _VaranDriveBase::GetParameterState
	VAR_INPUT
		us_Axis 	: USINT;
	END_VAR
	VAR_OUTPUT
		sd_para_state 	: DINT;
	END_VAR
  VAR
    p_Axis			: ^t_AxisData;
  END_VAR

	sd_para_state := -1;

	//look if class is ok
	if ( State <> _ClassOk ) & ( GetDriveIntState()$t_RtSSW <> CompGetSendParaList ) then
		return;
	end_if;

	//look if init was ok
	if ( b_InitOk ) then

		//------------------------------------------------------------------------------------------------
    //look which Axis we have and set pointers
//    if (us_Axis >= 0) & (us_Axis <= (AxisAvailableNo-1)) then
  if (us_Axis < DIASDRIVE_MAX_AXIS) & (aAxisData[us_Axis].e_AxisState <> _NotUsed) then
      p_Axis			:= #aAxisData[us_Axis];
    else
			sd_para_state := -2;
      return;
    end_if;

		//----------------------------------------------------------------------------------------------
		//look if Axis is in use
		if ( p_Axis^.e_AxisState = _NotUsed ) then
			sd_para_state := -3;
			return;
		end_if;

		//look if parameter handling is ready
		if	( p_Axis^.us_ParaReady	= _IdleState
			& p_Axis^.b_ListActive	= FALSE
			)
		then
			//look for an object handling error
      if (p_Axis^.sd_ObjectError = 0) then
        sd_para_state := 0;
      else
        sd_para_state := p_Axis^.sd_ObjectError;
      end_if;
		end_if;
	end_if;

END_FUNCTION

FUNCTION GLOBAL _VaranDriveBase::GetParameter
	VAR_INPUT
		us_Axis 	: USINT;
	END_VAR
	VAR_OUTPUT
		sd_para_data 	: DINT;
	END_VAR

	//get last object value of right Axis
//  if (us_Axis >= 0) & (us_Axis <= (AxisAvailableNo-1)) then
  if (us_Axis < DIASDRIVE_MAX_AXIS) & (aAxisData[us_Axis].e_AxisState <> _NotUsed) then
    sd_para_data := aAxisData[us_Axis].sd_Asyncdata;
  else
    sd_para_data := -1;
  end_if;

END_FUNCTION

FUNCTION GLOBAL _VaranDriveBase::SetParaList
	VAR_INPUT
		us_Axis 	: USINT;
		p_list 	: ^void;
		ui_counter 	: UINT;
	END_VAR
	VAR_OUTPUT
		sd_retval 	: DINT;
	END_VAR
  VAR
    p_Axis			: ^t_AxisData;
  END_VAR

	sd_retval := -1;

	//look if class is ok
	if ( State = _ClassOk ) | ( GetDriveIntState()$t_RtSSW = CompGetSendParaList ) then

    // if it's a SDD300 model
    if b_CompatibilityMode then
      //------------------------------------------------------------------------------------------------
      //look which Axis we have and set pointers
//      if (us_Axis >= 0) & (us_Axis <= (AxisAvailableNo-1)) then
      if (us_Axis < DIASDRIVE_MAX_AXIS) & (aAxisData[us_Axis].e_AxisState <> _NotUsed) then
        p_Axis        := #aAxisData[us_Axis];
      else
        sd_retval := -2;
        return;
      end_if;

      //-----------------------------------------------------------------------------------------------
      //look if Axis is in use
      if ( p_Axis^.e_AxisState = _NotUsed ) then
        sd_retval := -3;
        return;
      end_if;

      //-----------------------------------------------------------------------------------------------
      //look if we are in init or we can do it in realtime task

      //mark function as ok
      sd_retval := 0;

      //look if parameter handling is ready and list processing is active
      if	( p_Axis^.us_ParaReady = _IdleState
        & p_Axis^.b_ListActive = FALSE
        )
      then
        p_Axis^.p_ParaList$^void	:= p_list;
        p_Axis^.ui_ParaListCnt		:= ui_counter;

        // skip all defined parameter entries
        SkipEntries(us_Axis, p_Axis);

        //take over first parameter
        if ( p_Axis^.ui_ParaListCnt ) then
          IF SetParameter(us_Axis, p_Axis^.p_ParaList^.us_number, 1, p_Axis^.p_ParaList^.sd_value) = 0 THEN
            p_Axis^.b_ListActive		:= TRUE;
          p_Axis^.ui_ParaListCnt 	-= 1;
          p_Axis^.p_ParaList 		+= sizeof( t_ParaList );
          END_IF;
        end_if;

      else
        //not ready
        sd_retval := -1;
      end_if;
    else
    // if it's a SDD100/5000 model

      //------------------------------------------------------------------------------------------------
      //look which Axis we have and set pointers
//      if (us_Axis >= 0) & (us_Axis <= (AxisAvailableNo-1)) then
      if (us_Axis < DIASDRIVE_MAX_AXIS) & (aAxisData[us_Axis].e_AxisState <> _NotUsed) then
        p_Axis  := #aAxisData[us_Axis];
      else
        sd_retval := -2;
        return;
      end_if;

      //-----------------------------------------------------------------------------------------------
      //look if Axis is in use
      if ( p_Axis^.e_AxisState = _NotUsed ) then
        sd_retval := -3;
        return;
      end_if;

      //-----------------------------------------------------------------------------------------------
      //look if we are in init or we can do it in realtime task

      //mark function as ok
      sd_retval := 0;

      //look if parameter handling is ready and list processing is active
      if	( p_Axis^.us_ParaReady = _IdleState
        & p_Axis^.b_ListActive = FALSE
        )
      then
        p_Axis^.p_ParaList$^void	:= p_list;
        p_Axis^.ui_ParaListCnt		:= ui_counter;

        // skip all defined parameter entries
        SkipEntries(us_Axis, p_Axis);

        //take over first parameter
        if ( p_Axis^.ui_ParaListCnt ) then
          IF SetParameter(us_Axis, p_Axis^.p_ParaList^.us_number, 1, p_Axis^.p_ParaList^.sd_value) = 0 THEN
            p_Axis^.b_ListActive		:= TRUE;
          p_Axis^.ui_ParaListCnt 	-= 1;
          p_Axis^.p_ParaList 		+= sizeof( t_ParaList );
          END_IF;
        end_if;

      else
        //not ready
        sd_retval := -1;
      end_if;
    end_if;
  else
    //not ready
    sd_retval := -1;
  end_if;

END_FUNCTION

FUNCTION GLOBAL _VaranDriveBase::GetSyncParameter
	VAR_INPUT
		us_Axis 	: USINT;
		us_value 	: USINT;
		p_data 	: ^DINT;
	END_VAR
	VAR_OUTPUT
		sd_retval 	: DINT;
	END_VAR
  VAR
    p_Axis_data		: ^t_AxisData;
    sd_extend		: DINT;
  END_VAR

	//only if class is ok
	if ( State = _ClassOk ) then
    sd_retval := 0;

		//look for right value
		if ( us_value > 4 ) then
			sd_retval := -2;
			return;
		end_if;

    //look which Axis we have and set pointers
//    if (us_Axis >= 0) & (us_Axis <= (AxisAvailableNo-1)) then
    if (us_Axis < DIASDRIVE_MAX_AXIS) & (aAxisData[us_Axis].e_AxisState <> _NotUsed) then
      p_Axis_data			:= #aAxisData[us_Axis];
    else
      sd_retval := -3;
      return;
    end_if;

    sd_extend	:= aAxisData[us_Axis].b_ExtendedAxis;

		//only if Axis is ok
		if ( p_Axis_data^.e_AxisState = _AxisOk ) then

			//look if we have a extended value and extend mode is active else return
			if	( sd_extend	= 0 ) &
			    ( us_value  > 1 ) then

				sd_retval := -4;
				return;
			end_if;

			p_data^ := p_Axis_data^.s_ReadValues.a_SyncValues[ us_value ];
		end_if;
	else
		sd_retval := -1;
	end_if;

END_FUNCTION

FUNCTION GLOBAL _VaranDriveBase::SetSyncParameter
	VAR_INPUT
		us_Axis 	: USINT;
		us_value 	: USINT;
		sd_data 	: DINT;
	END_VAR
	VAR_OUTPUT
		sd_retval 	: DINT;
	END_VAR
  VAR
    p_Axis_data		: ^t_AxisData;
    sd_extend		: DINT;
  END_VAR

	//only if class is ok
	if ( State = _ClassOk ) then
    sd_retval := 0;

		//look for right value
		if ( us_value > 4 ) then
			sd_retval := -2;
			return;
		end_if;

    //look which Axis we have and set pointers
//    if (us_Axis >= 0) & (us_Axis <= (AxisAvailableNo-1)) then
    if (us_Axis < DIASDRIVE_MAX_AXIS) & (aAxisData[us_Axis].e_AxisState <> _NotUsed) then
      p_Axis_data			:= #aAxisData[us_Axis];
    else
      sd_retval := -3;
      return;
    end_if;

  	sd_extend	:= aAxisData[us_Axis].b_ExtendedAxis;

		//only if Axis is ok
		if ( p_Axis_data^.e_AxisState = _AxisOk ) then

			//look if we have a extended value and extend mode is active else return
			if	( sd_extend	= 0
				& us_value 	> 1
				)
			then

				sd_data := -4;
				return;
			end_if;

			p_Axis_data^.s_WriteValues.a_SyncValues[ us_value ] := sd_data;
		end_if;
	else
		sd_retval := -1;
	end_if;

END_FUNCTION

FUNCTION GLOBAL _VaranDriveBase::InitDrive
  VAR
    i : UDINT;
  END_VAR

	if ( b_InitOk ) then

		State := _NotInitialized;

    for i := 0 to (AxisAvailableNo-1) do
      if ( aAxisData[i].e_AxisState <> _NotUsed ) then
        aAxisData[i].e_AxisState := _NoInit;
      end_if;

      aAxisData[i].us_ParaReady := _IdleState;
    end_for;

		b_InitOk := 0;
    e_InitSSW:= _SetDataObjectOn;
    if b_CompatibilityMode = TRUE then
      e_RtSSW := CompInitAxis;
    else
      e_RtSSW := InitAxis;
    end_if;
	end_if;

END_FUNCTION

FUNCTION VIRTUAL GLOBAL _VaranDriveBase::SetDOsOff
  VAR
  	i : UDINT;
  END_VAR

  if AxisAvailableNo then
    // SDD300 model
    if b_CompatibilityMode then

      //disable data objects if Axis are used
      for i := 0 to (AxisAvailableNo-1) do
        if ( aAxisData[i].e_AxisState <> _NotUsed ) then
          DisableDO(ud_DOHandle:=aDataObjects[i].p_Handle$UDINT);
        end_if;
      end_for;
    else
    // SDD100/5000 model
      //disable data objects if Axis are used
      for i := 0 to (AxisAvailableNo-1) do
        if ( aAxisData[i].e_AxisState <> _NotUsed ) then
        DisableDO(ud_DOHandle:=newIsoDOs[i].p_Handle$UDINT);
        end_if;
      end_for;
      DisableDO(ud_DOHandle:=newAsyDO.p_Handle$UDINT);
    end_if;
  end_if;

  if newDigInDO.p_Handle then
    DisableDO(ud_DOHandle:=newDigInDO.p_Handle$UDINT);
  end_if;

(*
  //Fast Axis
  if ( UseFastAxis ) then
    s_DataFastAxis.p_Handle^.ucCtrlStat := VARAN_DO_NO_RUN;
  end_if;
*)
END_FUNCTION

FUNCTION VIRTUAL GLOBAL _VaranDriveBase::UpdateRetryCounter
  VAR
  	i : UDINT;
    tempRetryCounter : USINT;
  END_VAR

  // SDD300 model
  if b_CompatibilityMode then
    if CreatedCompDOs then
      //look for data object Axis
      if AxisAvailableNo then
        for i := 0 to (AxisAvailableNo-1) do
          if ( aAxisData[i].e_AxisState <> _NotUsed ) then
            tempRetryCounter := GetRetryCounter(ud_DOHandle := aDataObjects[i].p_Handle$UDINT);
            if ( tempRetryCounter <> aDataObjects[i].us_OldRetryCounter ) then
              RetryCounter += TO_USINT( tempRetryCounter - aDataObjects[i].us_OldRetryCounter );
              aDataObjects[i].us_OldRetryCounter := tempRetryCounter;
            end_if;
          end_if;
        end_for;
      end_if;
    end_if;
  else
    if CreatedNewIsoDOs then
    // SDD100/5000 model
      //look for data object Axis
      if AxisAvailableNo then
        for i := 0 to (AxisAvailableNo-1) do
          if ( aAxisData[i].e_AxisState <> _NotUsed ) then
            tempRetryCounter := GetRetryCounter(ud_DOHandle := newIsoDOs[i].p_Handle$UDINT);
            if ( tempRetryCounter <> newIsoDOs[i].us_OldRetryCounter ) then
              RetryCounter += TO_USINT( tempRetryCounter - newIsoDOs[i].us_OldRetryCounter );
              newIsoDOs[i].us_OldRetryCounter := tempRetryCounter;
            end_if;
          end_if;
        end_for;
      end_if;

      tempRetryCounter := GetRetryCounter(ud_DOHandle := newDigInDO.p_Handle$UDINT);
      if ( TempFetchDigitalInputs & (tempRetryCounter <> newDigInDO.us_OldRetryCounter) ) then
        RetryCounter += TO_USINT( tempRetryCounter - newDigInDO.us_OldRetryCounter );
        newDigInDO.us_OldRetryCounter := tempRetryCounter;
      end_if;
    end_if;
